KUKA KRL program: MyProgram_310().src

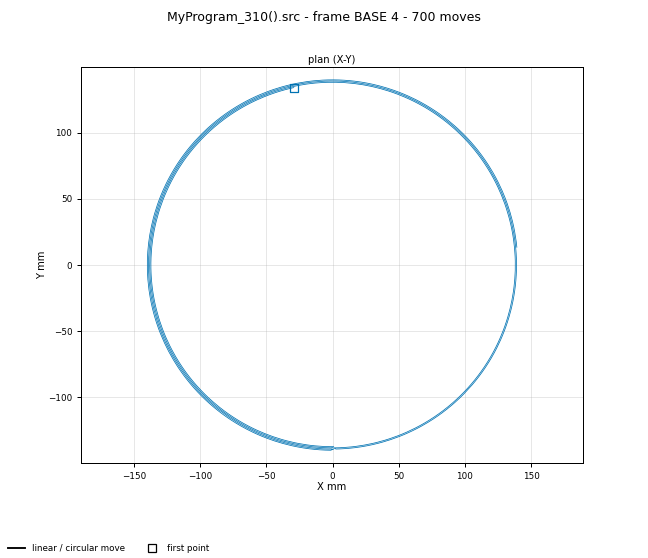
[picture p0: tool path of MyProgram_310().src in frame BASE 4, 700 of 700 moves have a stored position in this frame; points joined in program order, loops and branches not executed]
&ACCESS RVP
&REL 1
&PARAM TEMPLATE = C:\KRC\Roboter\Template\vorgabe
&PARAM EDITMASK = *
DEF MyProgram_310()
; ---- Setting reference (Base) ----
$BASE = BASE_DATA[4]

; --------------------------
; ---- Setting tool (TCP) ----
$TOOL = TOOL_DATA[3]
; --------------------------

$VEL.CP = VEL_APROX_PRINT
Startdeposition()
$VEL.CP = VEL_PRINT
LIN {X -29.2639,Y 134.0038,Z 182,A 103.6048,B 4.4109,C 0.0734,E1 4.3789,E2 349.3713} C_DIS
LIN {X -32.3216,Y 133.299,Z 182,A 104.9504,B 4.4109,C 0.0739,E1 4.3753,E2 348.0222} C_DIS
LIN {X -35.8759,Y 132.3877,Z 182,A 106.6346,B 4.4109,C 0.0736,E1 4.3707,E2 346.3204} C_DIS
LIN {X -40.2763,Y 131.1148,Z 182,A 108.4348,B 4.4108,C 0.076,E1 4.3659,E2 344.5352} C_DIS
LIN {X -43.6422,Y 130.0335,Z 182,A 110.3943,B 4.4108,C 0.0731,E1 4.3605,E2 342.5172} C_DIS
LIN {X -47.686,Y 128.606,Z 182,A 111.5731,B 4.4108,C 0.0799,E1 4.3576,E2 341.4149} C_DIS
LIN {X -51.93,Y 126.9528,Z 182,A 113.9515,B 4.4108,C 0.0778,E1 4.3513,E2 338.9794} C_DIS
LIN {X -54.9246,Y 125.6853,Z 182,A 115.0053,B 4.4107,C 0.0818,E1 4.3487,E2 337.964} C_DIS
LIN {X -57.8291,Y 124.3748,Z 182,A 116.3918,B 4.4107,C 0.0828,E1 4.3452,E2 336.5716} C_DIS
LIN {X -61.4347,Y 122.6365,Z 182,A 118.0932,B 4.4107,C 0.0846,E1 4.3409,E2 334.8678} C_DIS
LIN {X -64.5583,Y 121.0213,Z 182,A 119.5331,B 4.4106,C 0.0867,E1 4.3374,E2 333.4325} C_DIS
LIN {X -67.7824,Y 119.245,Z 182,A 121.2234,B 4.4106,C 0.0875,E1 4.3332,E2 331.7246} C_DIS
LIN {X -71.6244,Y 116.9775,Z 182,A 123.3545,B 4.4106,C 0.0881,E1 4.328,E2 329.5618} C_DIS
LIN {X -74.5849,Y 115.1125,Z 182,A 124.6005,B 4.4105,C 0.0919,E1 4.3252,E2 328.3436} C_DIS
LIN {X -78.3354,Y 112.5937,Z 182,A 126.5047,B 4.4105,C 0.0947,E1 4.3208,E2 326.4387} C_DIS
LIN {X -81.9968,Y 109.956,Z 182,A 128.4347,B 4.4104,C 0.0975,E1 4.3164,E2 324.5045} C_DIS
LIN {X -85.5745,Y 107.1952,Z 182,A 130.371,B 4.4103,C 0.1003,E1 4.3121,E2 322.5637} C_DIS
LIN {X -89.1427,Y 104.2473,Z 182,A 132.3771,B 4.4103,C 0.1033,E1 4.3078,E2 320.5502} C_DIS
LIN {X -92.5611,Y 101.2242,Z 182,A 134.3112,B 4.4101,C 0.1066,E1 4.3038,E2 318.6141} C_DIS
LIN {X -95.8331,Y 98.1319,Z 182,A 136.1996,B 4.4101,C 0.1102,E1 4.3,E2 316.7263} C_DIS
LIN {X -98.9014,Y 95.0391,Z 182,A 138.1181,B 4.41,C 0.1131,E1 4.2963,E2 314.7971} C_DIS
LIN {X -101.9762,Y 91.7318,Z 182,A 140.0414,B 4.4099,C 0.1167,E1 4.2926,E2 312.8707} C_DIS
LIN {X -104.9444,Y 88.3204,Z 182,A 141.957,B 4.4098,C 0.1206,E1 4.2891,E2 310.9533} C_DIS
LIN {X -107.7995,Y 84.8119,Z 182,A 143.9009,B 4.4097,C 0.1243,E1 4.2857,E2 309.0042} C_DIS
LIN {X -110.6043,Y 81.1202,Z 182,A 145.847,B 4.4096,C 0.1286,E1 4.2825,E2 307.0586} C_DIS
LIN {X -112.9805,Y 77.7767,Z 182,A 147.6562,B 4.4095,C 0.1319,E1 4.2796,E2 305.2389} C_DIS
LIN {X -115.8244,Y 73.475,Z 182,A 149.8731,B 4.4093,C 0.1366,E1 4.2762,E2 303.016} C_DIS
LIN {X -117.6466,Y 70.5207,Z 182,A 151.3055,B 4.4093,C 0.1402,E1 4.2741,E2 301.587} C_DIS
LIN {X -119.7774,Y 66.8381,Z 182,A 153.2138,B 4.4091,C 0.1437,E1 4.2715,E2 299.6639} C_DIS
LIN {X -121.98,Y 62.7249,Z 182,A 155.3274,B 4.409,C 0.1474,E1 4.2687,E2 297.5313} C_DIS
LIN {X -123.966,Y 58.7016,Z 182,A 157.0165,B 4.4088,C 0.1535,E1 4.2667,E2 295.8668} C_DIS
LIN {X -125.3677,Y 55.6446,Z 182,A 158.4571,B 4.4086,C 0.1568,E1 4.2651,E2 294.423} C_DIS
LIN {X -126.6541,Y 52.65,Z 182,A 159.7976,B 4.4086,C 0.1605,E1 4.2636,E2 293.0862} C_DIS
LIN {X -127.9591,Y 49.3944,Z 182,A 161.4133,B 4.4084,C 0.1634,E1 4.2619,E2 291.4528} C_DIS
LIN {X -130.0899,Y 43.4728,Z 182,A 164.1548,B 4.4082,C 0.1697,E1 4.2594,E2 288.6995} C_DIS
LIN {X -131.194,Y 40.0177,Z 182,A 166.0837,B 4.4082,C 0.171,E1 4.2578,E2 286.7197} C_DIS
LIN {X -132.3301,Y 36.0919,Z 182,A 167.3879,B 4.4078,C 0.1784,E1 4.2568,E2 285.4677} C_DIS
LIN {X -133.024,Y 33.4363,Z 182,A 168.6291,B 4.4078,C 0.1809,E1 4.256,E2 284.2155} C_DIS
LIN {X -133.8628,Y 29.9076,Z 182,A 170.2807,B 4.4076,C 0.1842,E1 4.2549,E2 282.548} C_DIS
LIN {X -134.7576,Y 25.568,Z 182,A 172.1099,B 4.4074,C 0.1895,E1 4.2539,E2 280.7228} C_DIS
LIN {X -135.4848,Y 21.3857,Z 182,A 173.9614,B 4.4072,C 0.1939,E1 4.2531,E2 278.863} C_DIS
LIN {X -135.9927,Y 17.8699,Z 182,A 175.4529,B 4.407,C 0.198,E1 4.2525,E2 277.3716} C_DIS
LIN {X -136.4492,Y 13.9804,Z 182,A 177.2549,B 4.4068,C 0.2016,E1 4.252,E2 275.5499} C_DIS
LIN {X -136.8021,Y 9.9275,Z 182,A 178.9425,B 4.4066,C 0.2064,E1 4.2516,E2 273.865} C_DIS
LIN {X -137.0448,Y 5.6759,Z 182,A -179.2169,B 4.4064,C 0.2111,E1 4.2513,E2 272.0179} C_DIS
LIN {X -137.1521,Y 1.7268,Z 182,A -177.4633,B 4.4062,C 0.2151,E1 4.2513,E2 270.2524} C_DIS
LIN {X -137.1387,Y -2.5339,Z 182,A -175.7226,B 4.4059,C 0.2204,E1 4.2513,E2 268.5179} C_DIS
LIN {X -137.0026,Y -6.6138,Z 182,A -173.9481,B 4.4057,C 0.2247,E1 4.2515,E2 266.7359} C_DIS
LIN {X -136.7867,Y -10.1386,Z 182,A -172.3669,B 4.4055,C 0.2282,E1 4.2518,E2 265.1422} C_DIS
LIN {X -136.3688,Y -14.7275,Z 182,A -170.4483,B 4.4052,C 0.2337,E1 4.2523,E2 263.2256} C_DIS
LIN {X -135.9713,Y -18.0329,Z 182,A -169.0247,B 4.4051,C 0.2373,E1 4.2528,E2 261.7988} C_DIS
LIN {X -135.4736,Y -21.4582,Z 182,A -167.5007,B 4.4049,C 0.2409,E1 4.2535,E2 260.2658} C_DIS
LIN {X -134.7446,Y -25.6362,Z 182,A -165.6181,B 4.4046,C 0.245,E1 4.2544,E2 258.3701} C_DIS
LIN {X -133.9141,Y -29.6793,Z 182,A -163.7588,B 4.4044,C 0.2489,E1 4.2555,E2 256.4946} C_DIS
LIN {X -132.9848,Y -33.5908,Z 182,A -162.1525,B 4.4041,C 0.254,E1 4.2566,E2 254.8986} C_DIS
LIN {X -131.3512,Y -39.504,Z 182,A -159.5891,B 4.4037,C 0.2609,E1 4.2585,E2 252.3367} C_DIS
LIN {X -130.4365,Y -42.4276,Z 182,A -158.0502,B 4.4037,C 0.2626,E1 4.2599,E2 250.7652} C_DIS
LIN {X -128.3433,Y -48.3872,Z 182,A -155.435,B 4.4032,C 0.2697,E1 4.2623,E2 248.1543} C_DIS
LIN {X -127.0767,Y -51.6226,Z 182,A -153.9839,B 4.403,C 0.2735,E1 4.2638,E2 246.704} C_DIS
LIN {X -125.713,Y -54.8607,Z 182,A -152.4663,B 4.4027,C 0.2769,E1 4.2655,E2 245.1807} C_DIS
LIN {X -124.3115,Y -57.9661,Z 182,A -150.9211,B 4.4026,C 0.2797,E1 4.2673,E2 243.6205} C_DIS
LIN {X -122.8733,Y -60.9546,Z 182,A -149.5531,B 4.4023,C 0.2832,E1 4.269,E2 242.2553} C_DIS
LIN {X -120.9706,Y -64.6528,Z 182,A -147.665,B 4.4021,C 0.2865,E1 4.2715,E2 240.3485} C_DIS
LIN {X -118.3587,Y -69.3183,Z 182,A -145.4078,B 4.4018,C 0.2917,E1 4.2746,E2 238.0892} C_DIS
LIN {X -116.1413,Y -72.9729,Z 182,A -143.5209,B 4.4016,C 0.2952,E1 4.2774,E2 236.1898} C_DIS
LIN {X -113.5739,Y -76.9074,Z 182,A -141.5681,B 4.4013,C 0.2998,E1 4.2804,E2 234.239} C_DIS
LIN {X -111.1027,Y -80.4362,Z 182,A -139.7071,B 4.401,C 0.3034,E1 4.2834,E2 232.3706} C_DIS
LIN {X -108.5628,Y -83.8329,Z 182,A -137.8763,B 4.4008,C 0.3068,E1 4.2866,E2 230.5326} C_DIS
LIN {X -105.8429,Y -87.2419,Z 182,A -135.969,B 4.4005,C 0.3101,E1 4.2899,E2 228.6148} C_DIS
LIN {X -102.8901,Y -90.7052,Z 182,A -133.4318,B 4.4006,C 0.3091,E1 4.2948,E2 225.9948} C_DIS
LIN {X -99.1771,Y -94.7506,Z 182,A -131.9418,B 4.3998,C 0.3199,E1 4.2974,E2 224.6103} C_DIS
LIN {X -96.5033,Y -97.4727,Z 182,A -130.2609,B 4.3997,C 0.3223,E1 4.3007,E2 222.9185} C_DIS
LIN {X -93.9205,Y -99.9639,Z 182,A -128.5538,B 4.3996,C 0.3235,E1 4.3042,E2 221.1845} C_DIS
LIN {X -90.6366,Y -102.9507,Z 182,A -126.441,B 4.3995,C 0.3247,E1 4.3087,E2 219.0381} C_DIS
LIN {X -88.135,Y -105.0999,Z 182,A -125.3023,B 4.3992,C 0.3291,E1 4.3111,E2 217.9309} C_DIS
LIN {X -85.5334,Y -107.2279,Z 182,A -123.8007,B 4.399,C 0.3306,E1 4.3144,E2 216.4166} C_DIS
LIN {X -81.9056,Y -110.0238,Z 182,A -121.8898,B 4.3988,C 0.3337,E1 4.3186,E2 214.5062} C_DIS
LIN {X -78.4854,Y -112.4894,Z 182,A -120.0573,B 4.3987,C 0.3359,E1 4.3228,E2 212.6644} C_DIS
LIN {X -74.8068,Y -114.9684,Z 182,A -118.1768,B 4.3985,C 0.3383,E1 4.3272,E2 210.7803} C_DIS
LIN {X -71.0909,Y -117.3025,Z 182,A -116.3724,B 4.3982,C 0.3411,E1 4.3315,E2 208.9797} C_DIS
LIN {X -67.5199,Y -119.3942,Z 182,A -114.5341,B 4.3982,C 0.3424,E1 4.336,E2 207.1269} C_DIS
LIN {X -63.7403,Y -121.4512,Z 182,A -112.8171,B 4.3979,C 0.3453,E1 4.3402,E2 205.4203} C_DIS
LIN {X -60.4027,Y -123.1455,Z 182,A -111.239,B 4.3978,C 0.347,E1 4.3442,E2 203.8401} C_DIS
LIN {X -57.3207,Y -124.6099,Z 182,A -109.8007,B 4.3977,C 0.3484,E1 4.3478,E2 202.3999} C_DIS
LIN {X -53.687,Y -126.2204,Z 182,A -108.1254,B 4.3976,C 0.35,E1 4.3521,E2 200.7225} C_DIS
LIN {X -51.231,Y -127.2345,Z 182,A -106.9551,B 4.3976,C 0.3505,E1 4.3551,E2 199.544} C_DIS
LIN {X -47.5863,Y -128.6433,Z 182,A -105.3745,B 4.3974,C 0.3524,E1 4.3593,E2 197.9699} C_DIS
LIN {X -44.8972,Y -129.6052,Z 182,A -104.1531,B 4.3974,C 0.3531,E1 4.3625,E2 196.7446} C_DIS
LIN {X -40.9503,Y -130.9084,Z 182,A -102.4109,B 4.3972,C 0.3543,E1 4.3671,E2 195.0012} C_DIS
LIN {X -38.449,Y -131.6623,Z 182,A -101.2729,B 4.3972,C 0.3546,E1 4.3702,E2 193.8567} C_DIS
LIN {X -34.9989,Y -132.6216,Z 182,A -99.7719,B 4.3972,C 0.3555,E1 4.3742,E2 192.3547} C_DIS
LIN {X -31.6937,Y -133.4504,Z 182,A -98.3727,B 4.397,C 0.3565,E1 4.378,E2 190.9583} C_DIS
LIN {X -28.7459,Y -134.1157,Z 182,A -97.1167,B 4.397,C 0.3571,E1 4.3815,E2 189.7027} C_DIS
LIN {X -25.5139,Y -134.768,Z 182,A -95.7025,B 4.397,C 0.3573,E1 4.3854,E2 188.2832} C_DIS
LIN {X -19.2093,Y -135.81,Z 182,A -93.1879,B 4.3968,C 0.3597,E1 4.3923,E2 185.7881} C_DIS
LIN {X -16.3537,Y -136.1834,Z 182,A -91.8444,B 4.3968,C 0.3586,E1 4.396,E2 184.4258} C_DIS
LIN {X -12.7776,Y -136.5657,Z 182,A -89.9841,B 4.3971,C 0.3552,E1 4.4013,E2 182.5175} C_DIS
LIN {X -9.1426,Y -136.8586,Z 182,A -88.7743,B 4.3969,C 0.3585,E1 4.4046,E2 181.3486} C_DIS
LIN {X -6.5538,Y -137.0056,Z 182,A -87.615,B 4.3969,C 0.3577,E1 4.4079,E2 180.1787} C_DIS
LIN {X -2.1717,Y -137.1447,Z 182,A -85.8504,B 4.3969,C 0.3582,E1 4.4128,E2 178.4221} C_DIS
LIN {X 0.9727,Y -137.1551,Z 182,A -84.8175,B 4.3967,C 0.3609,E1 4.4156,E2 177.4255} C_DIS
Enddeposition()
LIN {X 0.9727,Y -137.1551,Z 182,A -84.8175,B 4.3967,C 0.3609,E1 4.4156,E2 177.4255} C_DIS
Startdeposition()
$VEL.CP = VEL_PRINT
LIN {X -0.8195,Y -138.061,Z 182,A -85.9153,B 4.3834,C 0.3668,E1 4.3995,E2 178.6059} C_DIS
LIN {X -4.6066,Y -137.9886,Z 182,A -87.4496,B 4.3834,C 0.3665,E1 4.3952,E2 180.136} C_DIS
LIN {X -7.7094,Y -137.8501,Z 182,A -88.741,B 4.3834,C 0.3665,E1 4.3916,E2 181.4282} C_DIS
LIN {X -10.3826,Y -137.6727,Z 182,A -89.8567,B 4.3834,C 0.3665,E1 4.3885,E2 182.5448} C_DIS
LIN {X -13.4072,Y -137.4109,Z 182,A -91.1307,B 4.3834,C 0.3665,E1 4.3849,E2 183.8213} C_DIS
LIN {X -16.6884,Y -137.0513,Z 182,A -92.5339,B 4.3834,C 0.3665,E1 4.381,E2 185.2293} C_DIS
LIN {X -20.3271,Y -136.5609,Z 182,A -94.0261,B 4.3834,C 0.3658,E1 4.3769,E2 186.718} C_DIS
LIN {X -23.5214,Y -136.0471,Z 182,A -95.3761,B 4.3834,C 0.3654,E1 4.3732,E2 188.0694} C_DIS
LIN {X -26.161,Y -135.5621,Z 182,A -96.5101,B 4.3834,C 0.3652,E1 4.37,E2 189.2064} C_DIS
LIN {X -29.4753,Y -134.8804,Z 182,A -97.9114,B 4.3835,C 0.3645,E1 4.3662,E2 190.6077} C_DIS
LIN {X -33.1585,Y -134.0246,Z 182,A -99.4918,B 4.3836,C 0.3638,E1 4.3619,E2 192.1901} C_DIS
LIN {X -35.7982,Y -133.3414,Z 182,A -100.6484,B 4.3836,C 0.3634,E1 4.3588,E2 193.3503} C_DIS
LIN {X -39.0801,Y -132.4168,Z 182,A -102.0677,B 4.3837,C 0.3625,E1 4.355,E2 194.7704} C_DIS
LIN {X -42.3518,Y -131.4071,Z 182,A -103.5367,B 4.3837,C 0.3619,E1 4.351,E2 196.2461} C_DIS
LIN {X -46.0263,Y -130.1678,Z 182,A -105.1218,B 4.3839,C 0.3604,E1 4.3468,E2 197.8284} C_DIS
LIN {X -48.8301,Y -129.1401,Z 182,A -106.3786,B 4.3839,C 0.3595,E1 4.3435,E2 199.0878} C_DIS
LIN {X -52.4126,Y -127.7302,Z 182,A -107.9924,B 4.3841,C 0.3581,E1 4.3394,E2 200.7039} C_DIS
LIN {X -55.1251,Y -126.5808,Z 182,A -109.2309,B 4.3841,C 0.3571,E1 4.3362,E2 201.9447} C_DIS
LIN {X -58.2734,Y -125.1626,Z 182,A -110.6836,B 4.3843,C 0.3557,E1 4.3325,E2 203.4002} C_DIS
LIN {X -61.8592,Y -123.4323,Z 182,A -112.5047,B 4.3843,C 0.3553,E1 4.3279,E2 205.2436} C_DIS
LIN {X -65.7297,Y -121.4154,Z 182,A -114.2523,B 4.3845,C 0.3526,E1 4.3236,E2 206.983} C_DIS
LIN {X -69.3881,Y -119.3618,Z 182,A -116.0516,B 4.3847,C 0.3508,E1 4.3192,E2 208.7899} C_DIS
LIN {X -73.1029,Y -117.1234,Z 182,A -117.7965,B 4.3849,C 0.3479,E1 4.315,E2 210.5277} C_DIS
LIN {X -76.2241,Y -115.1169,Z 182,A -119.4346,B 4.385,C 0.3465,E1 4.3112,E2 212.1786} C_DIS
LIN {X -79.7324,Y -112.7149,Z 182,A -121.1604,B 4.3852,C 0.3435,E1 4.3072,E2 213.8993} C_DIS
LIN {X -82.8118,Y -110.473,Z 182,A -122.8802,B 4.3854,C 0.3421,E1 4.3033,E2 215.6372} C_DIS
LIN {X -86.3289,Y -107.747,Z 182,A -124.7605,B 4.3856,C 0.3393,E1 4.2992,E2 217.5217} C_DIS
LIN {X -89.7623,Y -104.9038,Z 182,A -126.598,B 4.3858,C 0.336,E1 4.2953,E2 219.3573} C_DIS
LIN {X -92.9151,Y -102.121,Z 182,A -128.3263,B 4.3861,C 0.3327,E1 4.2917,E2 221.0832} C_DIS
LIN {X -95.7133,Y -99.504,Z 182,A -130.0151,B 4.3862,C 0.3305,E1 4.2882,E2 222.7846} C_DIS
LIN {X -98.785,Y -96.4547,Z 182,A -131.8688,B 4.3865,C 0.3275,E1 4.2846,E2 224.6454} C_DIS
LIN {X -101.7729,Y -93.2963,Z 182,A -133.6694,B 4.3867,C 0.3239,E1 4.2811,E2 226.4451} C_DIS
LIN {X -104.3215,Y -90.4384,Z 182,A -135.3449,B 4.3869,C 0.3212,E1 4.278,E2 228.1314} C_DIS
LIN {X -107.1876,Y -87.0224,Z 182,A -137.2238,B 4.3872,C 0.3175,E1 4.2747,E2 230.0136} C_DIS
LIN {X -109.7812,Y -83.7258,Z 182,A -138.9788,B 4.3875,C 0.3138,E1 4.2717,E2 231.7698} C_DIS
LIN {X -112.2673,Y -80.3613,Z 182,A -140.8085,B 4.3877,C 0.3107,E1 4.2686,E2 233.6111} C_DIS
LIN {X -114.7245,Y -76.8128,Z 182,A -142.6406,B 4.388,C 0.3069,E1 4.2658,E2 235.4478} C_DIS
LIN {X -117.0649,Y -73.1968,Z 182,A -144.4981,B 4.3882,C 0.3032,E1 4.263,E2 237.3137} C_DIS
LIN {X -119.267,Y -69.5519,Z 182,A -146.2815,B 4.3885,C 0.2991,E1 4.2604,E2 239.0986} C_DIS
LIN {X -121.4154,Y -65.7297,Z 182,A -148.2159,B 4.3887,C 0.2955,E1 4.2578,E2 241.047} C_DIS
LIN {X -123.2037,Y -62.3081,Z 182,A -149.74,B 4.389,C 0.2909,E1 4.2558,E2 242.5603} C_DIS
LIN {X -124.9503,Y -58.7325,Z 182,A -151.4376,B 4.3893,C 0.2871,E1 4.2538,E2 244.2632} C_DIS
LIN {X -126.2793,Y -55.8143,Z 182,A -152.7859,B 4.3895,C 0.2838,E1 4.2522,E2 245.613} C_DIS
LIN {X -127.5386,Y -52.8713,Z 182,A -154.1755,B 4.3897,C 0.2808,E1 4.2507,E2 247.0099} C_DIS
LIN {X -128.8126,Y -49.687,Z 182,A -155.6413,B 4.3899,C 0.2774,E1 4.2492,E2 248.4803} C_DIS
LIN {X -130.001,Y -46.489,Z 182,A -157.1006,B 4.3901,C 0.274,E1 4.2478,E2 249.9445} C_DIS
LIN {X -131.0722,Y -43.3763,Z 182,A -158.5205,B 4.3903,C 0.2707,E1 4.2465,E2 251.3705} C_DIS
LIN {X -132.2647,Y -39.5998,Z 182,A -160.2028,B 4.3906,C 0.2665,E1 4.2452,E2 253.057} C_DIS
LIN {X -133.1864,Y -36.3794,Z 182,A -161.6362,B 4.3908,C 0.2631,E1 4.2441,E2 254.495} C_DIS
LIN {X -133.8647,Y -33.7887,Z 182,A -162.7816,B 4.391,C 0.2603,E1 4.2433,E2 255.6441} C_DIS
LIN {X -134.6625,Y -30.4548,Z 182,A -164.2614,B 4.3912,C 0.2567,E1 4.2423,E2 257.1304} C_DIS
LIN {X -135.4539,Y -26.7266,Z 182,A -165.8816,B 4.3914,C 0.2526,E1 4.2414,E2 258.7546} C_DIS
LIN {X -135.9643,Y -23.9842,Z 182,A -167.0752,B 4.3916,C 0.2497,E1 4.2408,E2 259.952} C_DIS
LIN {X -136.4895,Y -20.7882,Z 182,A -168.4619,B 4.3918,C 0.2462,E1 4.2402,E2 261.3432} C_DIS
LIN {X -136.9365,Y -17.6054,Z 182,A -169.8781,B 4.3919,C 0.243,E1 4.2397,E2 262.769} C_DIS
LIN {X -137.3066,Y -14.4381,Z 182,A -171.204,B 4.3921,C 0.2393,E1 4.2393,E2 264.0944} C_DIS
LIN {X -137.5888,Y -11.4373,Z 182,A -172.5095,B 4.3923,C 0.2361,E1 4.239,E2 265.4059} C_DIS
LIN {X -137.8075,Y -8.4003,Z 182,A -173.8339,B 4.3925,C 0.233,E1 4.2387,E2 266.7372} C_DIS
LIN {X -137.9712,Y -5.0541,Z 182,A -175.2723,B 4.3927,C 0.2293,E1 4.2385,E2 268.1807} C_DIS
LIN {X -138.0618,Y -0.8135,Z 182,A -177.0703,B 4.3929,C 0.2246,E1 4.2385,E2 269.9822} C_DIS
LIN {X -138.0434,Y 2.3508,Z 182,A -178.4274,B 4.3931,C 0.2212,E1 4.2385,E2 271.3439} C_DIS
LIN {X -137.9448,Y 5.7297,Z 182,A -179.9008,B 4.3933,C 0.2177,E1 4.2386,E2 272.8252} C_DIS
LIN {X -137.754,Y 9.2695,Z 182,A 178.6109,B 4.3935,C 0.2136,E1 4.2389,E2 274.3147} C_DIS
LIN {X -137.5453,Y 11.9519,Z 182,A 177.4146,B 4.3935,C 0.211,E1 4.2392,E2 275.5201} C_DIS
LIN {X -137.0709,Y 16.5243,Z 182,A 175.4536,B 4.3938,C 0.2059,E1 4.2398,E2 277.4863} C_DIS
LIN {X -136.6041,Y 20.0248,Z 182,A 173.9413,B 4.394,C 0.2021,E1 4.2404,E2 279.0034} C_DIS
LIN {X -136.0471,Y 23.5214,Z 182,A 172.439,B 4.3942,C 0.1982,E1 4.241,E2 280.5088} C_DIS
LIN {X -135.4539,Y 26.7266,Z 182,A 171.0385,B 4.3943,C 0.1948,E1 4.2418,E2 281.9142} C_DIS
LIN {X -134.905,Y 29.3618,Z 182,A 169.8668,B 4.3945,C 0.192,E1 4.2425,E2 283.0918} C_DIS
LIN {X -134.0246,Y 33.1585,Z 182,A 168.209,B 4.3946,C 0.1878,E1 4.2435,E2 284.7535} C_DIS
LIN {X -133.3105,Y 35.914,Z 182,A 166.9863,B 4.3948,C 0.1849,E1 4.2444,E2 285.9803} C_DIS
LIN {X -132.4154,Y 39.0851,Z 182,A 165.5801,B 4.3949,C 0.1814,E1 4.2455,E2 287.3902} C_DIS
LIN {X -131.4071,Y 42.3518,Z 182,A 164.0634,B 4.395,C 0.1782,E1 4.2468,E2 288.918} C_DIS
LIN {X -130.1678,Y 46.0263,Z 182,A 162.4427,B 4.3952,C 0.174,E1 4.2483,E2 290.5389} C_DIS
LIN {X -128.9918,Y 49.2261,Z 182,A 160.9811,B 4.3953,C 0.1705,E1 4.2497,E2 292.0052} C_DIS
LIN {X -127.7302,Y 52.4126,Z 182,A 159.5121,B 4.3955,C 0.1671,E1 4.2512,E2 293.4789} C_DIS
LIN {X -126.602,Y 55.0761,Z 182,A 158.2661,B 4.3955,C 0.1643,E1 4.2526,E2 294.7295} C_DIS
LIN {X -125.1604,Y 58.2781,Z 182,A 156.7688,B 4.3957,C 0.1608,E1 4.2544,E2 296.2306} C_DIS
LIN {X -123.6547,Y 61.4083,Z 182,A 155.2388,B 4.3958,C 0.1577,E1 4.2563,E2 297.7703} C_DIS
LIN {X -121.7097,Y 65.1819,Z 182,A 153.3744,B 4.396,C 0.154,E1 4.2587,E2 299.6461} C_DIS
LIN {X -119.5507,Y 69.0619,Z 182,A 151.4737,B 4.396,C 0.1499,E1 4.2613,E2 301.5523} C_DIS
LIN {X -117.4547,Y 72.5706,Z 182,A 149.8211,B 4.3962,C 0.1455,E1 4.2637,E2 303.1982} C_DIS
LIN {X -115.2806,Y 75.9755,Z 182,A 148.0718,B 4.3964,C 0.142,E1 4.2664,E2 304.9551} C_DIS
LIN {X -112.9675,Y 79.3744,Z 182,A 146.2555,B 4.3964,C 0.1388,E1 4.2693,E2 306.7836} C_DIS
LIN {X -110.6264,Y 82.6058,Z 182,A 144.6421,B 4.3966,C 0.1348,E1 4.2719,E2 308.3903} C_DIS
LIN {X -108.3017,Y 85.632,Z 182,A 142.9232,B 4.3966,C 0.1322,E1 4.2749,E2 310.1247} C_DIS
LIN {X -105.4817,Y 89.0826,Z 182,A 141.0517,B 4.3968,C 0.1284,E1 4.2782,E2 311.9974} C_DIS
LIN {X -102.7198,Y 92.2526,Z 182,A 139.2931,B 4.3968,C 0.1248,E1 4.2815,E2 313.7562} C_DIS
LIN {X -99.7357,Y 95.4709,Z 182,A 137.3865,B 4.397,C 0.1217,E1 4.2852,E2 315.6718} C_DIS
LIN {X -96.5396,Y 98.7017,Z 182,A 135.5306,B 4.397,C 0.1178,E1 4.2888,E2 317.5225} C_DIS
LIN {X -93.7638,Y 101.3431,Z 182,A 133.9043,B 4.3971,C 0.115,E1 4.2921,E2 319.152} C_DIS
LIN {X -91.1109,Y 103.7347,Z 182,A 132.3179,B 4.3971,C 0.113,E1 4.2955,E2 320.75} C_DIS
LIN {X -87.8397,Y 106.5183,Z 182,A 130.4861,B 4.3973,C 0.1102,E1 4.2994,E2 322.5864} C_DIS
LIN {X -84.4316,Y 109.2393,Z 182,A 128.6902,B 4.3973,C 0.107,E1 4.3033,E2 324.3792} C_DIS
LIN {X -81.3829,Y 111.5299,Z 182,A 127.0473,B 4.3974,C 0.1049,E1 4.307,E2 326.0283} C_DIS
LIN {X -77.9699,Y 113.9413,Z 182,A 125.3115,B 4.3974,C 0.1021,E1 4.311,E2 327.7629} C_DIS
LIN {X -74.8095,Y 116.0414,Z 182,A 123.7393,B 4.3975,C 0.0997,E1 4.3147,E2 329.3337} C_DIS
LIN {X -71.2836,Y 118.2395,Z 182,A 121.9574,B 4.3975,C 0.0977,E1 4.319,E2 331.1213} C_DIS
LIN {X -67.8083,Y 120.2662,Z 182,A 120.1905,B 4.3975,C 0.0962,E1 4.3233,E2 332.899} C_DIS
LIN {X -63.8596,Y 122.4067,Z 182,A 118.4046,B 4.3977,C 0.0932,E1 4.3276,E2 334.6739} C_DIS
LIN {X -60.2989,Y 124.2019,Z 182,A 116.7273,B 4.3977,C 0.0914,E1 4.3318,E2 336.3529} C_DIS
LIN {X -57.4185,Y 125.5579,Z 182,A 115.375,B 4.3977,C 0.0901,E1 4.3353,E2 337.7081} C_DIS
LIN {X -54.382,Y 126.9021,Z 182,A 114.0038,B 4.3977,C 0.0886,E1 4.3388,E2 339.0775} C_DIS
LIN {X -51.2811,Y 128.1863,Z 182,A 112.5879,B 4.3977,C 0.0874,E1 4.3424,E2 340.4952} C_DIS
LIN {X -48.0895,Y 129.4175,Z 182,A 111.1542,B 4.3978,C 0.0861,E1 4.3462,E2 341.9297} C_DIS
LIN {X -44.8859,Y 130.5632,Z 182,A 109.7298,B 4.3978,C 0.085,E1 4.35,E2 343.3548} C_DIS
LIN {X -41.4038,Y 131.7099,Z 182,A 108.1872,B 4.3978,C 0.084,E1 4.3541,E2 344.899} C_DIS
LIN {X -37.9899,Y 132.736,Z 182,A 106.7053,B 4.3978,C 0.0829,E1 4.358,E2 346.3804} C_DIS
LIN {X -35.1003,Y 133.5275,Z 182,A 105.4796,B 4.3978,C 0.0819,E1 4.3613,E2 347.6031} C_DIS
LIN {X -32.0139,Y 134.3005,Z 182,A 104.0866,B 4.3978,C 0.0817,E1 4.3651,E2 349.0042} C_DIS
LIN {X -28.3324,Y 135.1272,Z 182,A 102.5528,B 4.3979,C 0.0806,E1 4.3693,E2 350.5333} C_DIS
LIN {X -25.5863,Y 135.6719,Z 182,A 101.3868,B 4.3979,C 0.0801,E1 4.3725,E2 351.699} C_DIS
LIN {X -22.3847,Y 136.2368,Z 182,A 100.0333,B 4.3979,C 0.0796,E1 4.3762,E2 353.0523} C_DIS
LIN {X -19.195,Y 136.7227,Z 182,A 98.6914,B 4.3979,C 0.0791,E1 4.3799,E2 354.3939} C_DIS
LIN {X -15.5617,Y 137.1857,Z 182,A 97.1686,B 4.3979,C 0.0787,E1 4.3842,E2 355.9164} C_DIS
LIN {X -12.8611,Y 137.4633,Z 182,A 96.022,B 4.3979,C 0.0787,E1 4.3874,E2 357.0647} C_DIS
LIN {X -9.2695,Y 137.754,Z 182,A 94.5461,B 4.3979,C 0.0783,E1 4.3915,E2 358.5376} C_DIS
LIN {X -6.6042,Y 137.9057,Z 182,A 93.4663,B 4.3979,C 0.0779,E1 4.3945,E2 359.6134} C_DIS
LIN {X -3.9025,Y 138.0082,Z 182,A 92.2784,B 4.3979,C 0.0785,E1 4.3978,E2 360.8088} C_DIS
LIN {X 0,Y 138.0655,Z 182,A 90.7024,B 4.3979,C 0.0782,E1 4.4022,E2 362.3789} C_DIS
LIN {X 2.6207,Y 138.0389,Z 182,A 89.5769,B 4.3979,C 0.0787,E1 4.4053,E2 363.5085} C_DIS
LIN {X 6.155,Y 137.9282,Z 182,A 88.1464,B 4.3979,C 0.0786,E1 4.4093,E2 364.9339} C_DIS
LIN {X 9.2695,Y 137.754,Z 182,A 86.8533,B 4.3979,C 0.0789,E1 4.4129,E2 366.2263} C_DIS
LIN {X 13.9815,Y 137.3557,Z 182,A 84.8946,B 4.3979,C 0.0795,E1 4.4184,E2 368.1839} C_DIS
LIN {X 16.6884,Y 137.0513,Z 182,A 83.7284,B 4.3979,C 0.0803,E1 4.4216,E2 369.3539} C_DIS
LIN {X 20.3271,Y 136.5609,Z 182,A 82.2489,B 4.3979,C 0.0805,E1 4.4257,E2 370.8276} C_DIS
LIN {X 22.9824,Y 136.1371,Z 182,A 81.0868,B 4.3979,C 0.0816,E1 4.4289,E2 371.995} C_DIS
LIN {X 26.7266,Y 135.4539,Z 182,A 79.5665,B 4.3979,C 0.0819,E1 4.4331,E2 373.5076} C_DIS
LIN {X 29.4753,Y 134.8804,Z 182,A 78.4076,B 4.3979,C 0.0826,E1 4.4362,E2 374.6653} C_DIS
LIN {X 33.0405,Y 134.053,Z 182,A 76.9042,B 4.3979,C 0.0836,E1 4.4403,E2 376.1665} C_DIS
LIN {X 35.914,Y 133.3105,Z 182,A 75.677,B 4.3979,C 0.0845,E1 4.4436,E2 377.3929} C_DIS
LIN {X 39.1345,Y 132.4009,Z 182,A 74.2999,B 4.3979,C 0.0855,E1 4.4473,E2 378.7681} C_DIS
LIN {X 42.3518,Y 131.4071,Z 182,A 72.8751,B 4.3978,C 0.0871,E1 4.4511,E2 380.196} C_DIS
LIN {X 45.7133,Y 130.2763,Z 182,A 71.4551,B 4.3978,C 0.088,E1 4.4549,E2 381.6094} C_DIS
LIN {X 49.2261,Y 128.9918,Z 182,A 69.9231,B 4.3978,C 0.0894,E1 4.4589,E2 383.1387} C_DIS
LIN {X 52.4126,Y 127.7302,Z 182,A 68.5172,B 4.3978,C 0.0908,E1 4.4625,E2 384.5424} C_DIS
LIN {X 55.0623,Y 126.608,Z 182,A 67.3295,B 4.3977,C 0.0922,E1 4.4656,E2 385.7291} C_DIS
LIN {X 58.2781,Y 125.1604,Z 182,A 65.8932,B 4.3977,C 0.0937,E1 4.4692,E2 387.162} C_DIS
LIN {X 61.8592,Y 123.4323,Z 182,A 64.1239,B 4.3976,C 0.0971,E1 4.4737,E2 388.9458} C_DIS
LIN {X 65.7297,Y 121.4154,Z 182,A 62.3567,B 4.3976,C 0.0991,E1 4.478,E2 390.7074} C_DIS
LIN {X 69.5519,Y 119.267,Z 182,A 60.691,B 4.3976,C 0.1001,E1 4.482,E2 392.3542} C_DIS
LIN {X 72.5706,Y 117.4547,Z 182,A 59.2411,B 4.3975,C 0.1022,E1 4.4855,E2 393.8028} C_DIS
LIN {X 76.076,Y 115.2144,Z 182,A 57.5258,B 4.3975,C 0.1048,E1 4.4895,E2 395.5167} C_DIS
LIN {X 79.217,Y 113.0785,Z 182,A 55.939,B 4.3973,C 0.1075,E1 4.4931,E2 397.1048} C_DIS
LIN {X 82.8118,Y 110.473,Z 182,A 54.1417,B 4.3973,C 0.1102,E1 4.4972,E2 398.8967} C_DIS
LIN {X 86.2542,Y 107.8064,Z 182,A 52.3605,B 4.3972,C 0.1131,E1 4.5011,E2 400.6748} C_DIS
LIN {X 89.6532,Y 104.9966,Z 182,A 50.5624,B 4.3972,C 0.1161,E1 4.5049,E2 402.4692} C_DIS
LIN {X 92.9151,Y 102.121,Z 182,A 48.8415,B 4.3971,C 0.1186,E1 4.5085,E2 404.18} C_DIS
LIN {X 95.8988,Y 99.3244,Z 182,A 47.1188,B 4.397,C 0.1223,E1 4.512,E2 405.9061} C_DIS
LIN {X 99.1246,Y 96.1051,Z 182,A 45.2833,B 4.3969,C 0.1255,E1 4.5155,E2 407.735} C_DIS
LIN {X 101.9476,Y 93.1062,Z 182,A 43.5891,B 4.3968,C 0.1289,E1 4.5188,E2 409.4277} C_DIS
LIN {X 104.9038,Y 89.7623,Z 182,A 41.8136,B 4.3967,C 0.132,E1 4.522,E2 411.1942} C_DIS
LIN {X 107.5853,Y 86.5293,Z 182,A 40.1606,B 4.3966,C 0.1348,E1 4.5249,E2 412.8364} C_DIS
LIN {X 109.9374,Y 83.5216,Z 182,A 38.5603,B 4.3965,C 0.1386,E1 4.5276,E2 414.4392} C_DIS
LIN {X 112.5672,Y 79.9419,Z 182,A 36.854,B 4.3964,C 0.1412,E1 4.5304,E2 416.1289} C_DIS
LIN {X 114.7245,Y 76.8128,Z 182,A 35.2409,B 4.3963,C 0.1453,E1 4.5329,E2 417.747} C_DIS
LIN {X 117.1234,Y 73.1029,Z 182,A 33.4702,B 4.3961,C 0.149,E1 4.5356,E2 419.5105} C_DIS
LIN {X 119.267,Y 69.5519,Z 182,A 31.8045,B 4.3961,C 0.1525,E1 4.5379,E2 421.17} C_DIS
LIN {X 121.4154,Y 65.7297,Z 182,A 29.9777,B 4.3958,C 0.1571,E1 4.5404,E2 422.9984} C_DIS
LIN {X 123.2037,Y 62.3081,Z 182,A 28.5009,B 4.3958,C 0.1596,E1 4.5423,E2 424.4601} C_DIS
LIN {X 124.9503,Y 58.7325,Z 182,A 26.9385,B 4.3956,C 0.1627,E1 4.5442,E2 426.0121} C_DIS
LIN {X 126.383,Y 55.5825,Z 182,A 25.5455,B 4.3956,C 0.1659,E1 4.5457,E2 427.4004} C_DIS
LIN {X 127.5386,Y 52.8713,Z 182,A 24.3598,B 4.3954,C 0.1686,E1 4.547,E2 428.5819} C_DIS
LIN {X 128.8126,Y 49.687,Z 182,A 22.9805,B 4.3953,C 0.1718,E1 4.5484,E2 429.9563} C_DIS
LIN {X 129.9939,Y 46.5087,Z 182,A 21.6144,B 4.3952,C 0.1751,E1 4.5497,E2 431.318} C_DIS
LIN {X 131.1041,Y 43.2805,Z 182,A 20.2053,B 4.395,C 0.1788,E1 4.551,E2 432.7269} C_DIS
LIN {X 132.2489,Y 39.6512,Z 182,A 18.7189,B 4.3949,C 0.1819,E1 4.5522,E2 434.2025} C_DIS
LIN {X 133.0573,Y 36.8411,Z 182,A 17.5024,B 4.3948,C 0.1852,E1 4.5531,E2 435.42} C_DIS
LIN {X 133.9065,Y 33.6238,Z 182,A 16.2037,B 4.3946,C 0.188,E1 4.554,E2 436.709} C_DIS
LIN {X 134.7801,Y 29.9399,Z 182,A 14.683,B 4.3945,C 0.1917,E1 4.555,E2 438.2244} C_DIS
LIN {X 135.4539,Y 26.7266,Z 182,A 13.3647,B 4.3943,C 0.1949,E1 4.5557,E2 439.5379} C_DIS
LIN {X 136.2368,Y 22.3847,Z 182,A 11.5943,B 4.3941,C 0.1992,E1 4.5565,E2 441.3016} C_DIS
LIN {X 136.7227,Y 19.195,Z 182,A 10.2997,B 4.394,C 0.2024,E1 4.5571,E2 442.5915} C_DIS
LIN {X 137.1857,Y 15.5617,Z 182,A 8.8294,B 4.3938,C 0.2061,E1 4.5576,E2 444.0565} C_DIS
LIN {X 137.4633,Y 12.8611,Z 182,A 7.7525,B 4.3938,C 0.2086,E1 4.5579,E2 445.1278} C_DIS
LIN {X 137.754,Y 9.2695,Z 182,A 6.2948,B 4.3935,C 0.2123,E1 4.5582,E2 446.5818} C_DIS
LIN {X 137.9057,Y 6.6042,Z 182,A 5.2247,B 4.3935,C 0.215,E1 4.5583,E2 447.6478} C_DIS
LIN {X 138.0315,Y 3.0645,Z 182,A 3.6488,B 4.3931,C 0.2205,E1 4.5584,E2 449.2382} C_DIS
LIN {X 138.0618,Y -0.8135,Z 182,A 2.1458,B 4.393,C 0.2237,E1 4.5584,E2 450.7287} C_DIS
LIN {X 138.004,Y -4.0532,Z 182,A 0.8886,B 4.3928,C 0.2264,E1 4.5584,E2 451.9758} C_DIS
LIN {X 137.8501,Y -7.7094,Z 182,A -0.5322,B 4.3927,C 0.2294,E1 4.5582,E2 453.3852} C_DIS
LIN {X 137.6727,Y -10.3826,Z 182,A -1.6118,B 4.3925,C 0.2322,E1 4.558,E2 454.4615} C_DIS
LIN {X 137.3557,Y -13.9815,Z 182,A -3.0654,B 4.3923,C 0.2358,E1 4.5576,E2 455.9104} C_DIS
LIN {X 137.0652,Y -16.5719,Z 182,A -4.1705,B 4.3922,C 0.2392,E1 4.5572,E2 457.0192} C_DIS
LIN {X 136.5609,Y -20.3271,Z 182,A -5.6407,B 4.392,C 0.2423,E1 4.5566,E2 458.4776} C_DIS
LIN {X 136.0471,Y -23.5214,Z 182,A -6.9434,B 4.3918,C 0.2455,E1 4.5561,E2 459.7762} C_DIS
LIN {X 135.4539,Y -26.7266,Z 182,A -8.2561,B 4.3916,C 0.2488,E1 4.5554,E2 461.0849} C_DIS
LIN {X 134.9226,Y -29.28,Z 182,A -9.3234,B 4.3915,C 0.2516,E1 4.5547,E2 462.151} C_DIS
LIN {X 134.0658,Y -32.9876,Z 182,A -10.845,B 4.3913,C 0.2553,E1 4.5538,E2 463.6665} C_DIS
LIN {X 133.3105,Y -35.914,Z 182,A -12.0567,B 4.3911,C 0.2582,E1 4.5529,E2 464.8737} C_DIS
LIN {X 132.4009,Y -39.1345,Z 182,A -13.4046,B 4.3909,C 0.2614,E1 4.5519,E2 466.2175} C_DIS
LIN {X 131.4071,Y -42.3518,Z 182,A -14.8004,B 4.3907,C 0.2652,E1 4.5507,E2 467.6142} C_DIS
LIN {X 130.1678,Y -46.0263,Z 182,A -16.3234,B 4.3905,C 0.2685,E1 4.5493,E2 469.1275} C_DIS
LIN {X 128.9918,Y -49.2261,Z 182,A -17.6975,B 4.3903,C 0.2717,E1 4.548,E2 470.4974} C_DIS
LIN {X 127.7302,Y -52.4126,Z 182,A -19.0792,B 4.3901,C 0.275,E1 4.5465,E2 471.8751} C_DIS
LIN {X 126.6172,Y -55.0409,Z 182,A -20.241,B 4.3899,C 0.2778,E1 4.5453,E2 473.0349} C_DIS
LIN {X 125.1604,Y -58.2781,Z 182,A -21.6618,B 4.3897,C 0.281,E1 4.5436,E2 474.4502} C_DIS
LIN {X 123.4323,Y -61.8592,Z 182,A -23.405,B 4.3893,C 0.2865,E1 4.5414,E2 476.2069} C_DIS
LIN {X 121.447,Y -65.6708,Z 182,A -25.0776,B 4.3891,C 0.2896,E1 4.5393,E2 477.8667} C_DIS
LIN {X 119.267,Y -69.5519,Z 182,A -26.8559,B 4.3889,C 0.2933,E1 4.5368,E2 479.6376} C_DIS
LIN {X 117.1234,Y -73.1029,Z 182,A -28.5253,B 4.3886,C 0.2969,E1 4.5344,E2 481.3017} C_DIS
LIN {X 114.683,Y -76.875,Z 182,A -30.3672,B 4.3883,C 0.3011,E1 4.5316,E2 483.1423} C_DIS
LIN {X 112.2002,Y -80.4552,Z 182,A -32.0473,B 4.3882,C 0.3038,E1 4.5289,E2 484.8072} C_DIS
LIN {X 110.0922,Y -83.3165,Z 182,A -33.5158,B 4.3879,C 0.3072,E1 4.5264,E2 486.2762} C_DIS
LIN {X 107.5513,Y -86.5714,Z 182,A -35.2442,B 4.3876,C 0.3113,E1 4.5234,E2 488.0079} C_DIS
LIN {X 104.9038,Y -89.7623,Z 182,A -36.8927,B 4.3874,C 0.3142,E1 4.5205,E2 489.6485} C_DIS
LIN {X 102.121,Y -92.9151,Z 182,A -38.5351,B 4.3873,C 0.3167,E1 4.5174,E2 491.279} C_DIS
LIN {X 99.504,Y -95.7133,Z 182,A -40.1475,B 4.387,C 0.3204,E1 4.5143,E2 492.8956} C_DIS
LIN {X 96.5396,Y -98.7017,Z 182,A -41.793,B 4.3868,C 0.3228,E1 4.5111,E2 494.5294} C_DIS
LIN {X 93.7638,Y -101.3431,Z 182,A -43.4074,B 4.3866,C 0.3263,E1 4.5078,E2 496.1483} C_DIS
LIN {X 90.6327,Y -104.1519,Z 182,A -45.0855,B 4.3864,C 0.3289,E1 4.5043,E2 497.8189} C_DIS
LIN {X 87.4736,Y -106.8189,Z 182,A -46.8229,B 4.3861,C 0.3324,E1 4.5006,E2 499.5606} C_DIS
LIN {X 83.9733,Y -109.5919,Z 182,A -48.6343,B 4.3859,C 0.3353,E1 4.4966,E2 501.368} C_DIS
LIN {X 80.4552,Y -112.2002,Z 182,A -50.4085,B 4.3857,C 0.338,E1 4.4926,E2 503.138} C_DIS
LIN {X 76.8128,Y -114.7245,Z 182,A -52.2141,B 4.3855,C 0.3407,E1 4.4884,E2 504.9407} C_DIS
LIN {X 73.1029,Y -117.1234,Z 182,A -53.995,B 4.3853,C 0.343,E1 4.4842,E2 506.7162} C_DIS
LIN {X 69.5519,Y -119.267,Z 182,A -55.6778,B 4.3851,C 0.3453,E1 4.4802,E2 508.3953} C_DIS
LIN {X 65.7297,Y -121.4154,Z 182,A -57.5255,B 4.3849,C 0.3483,E1 4.4757,E2 510.248} C_DIS
LIN {X 62.3081,Y -123.2037,Z 182,A -59.0215,B 4.3848,C 0.3493,E1 4.472,E2 511.7312} C_DIS
LIN {X 58.7325,Y -124.9503,Z 182,A -60.6057,B 4.3847,C 0.3507,E1 4.468,E2 513.3079} C_DIS
LIN {X 56.0831,Y -126.1591,Z 182,A -61.8011,B 4.3846,C 0.3521,E1 4.465,E2 514.5023} C_DIS
LIN {X 52.8713,Y -127.5386,Z 182,A -63.2243,B 4.3844,C 0.3536,E1 4.4613,E2 515.923} C_DIS
LIN {X 49.687,Y -128.8126,Z 182,A -64.6269,B 4.3844,C 0.355,E1 4.4577,E2 517.3239} C_DIS
LIN {X 46.489,Y -130.001,Z 182,A -66.0239,B 4.3842,C 0.3563,E1 4.454,E2 518.7194} C_DIS
LIN {X 43.2805,Y -131.1041,Z 182,A -67.428,B 4.3842,C 0.3577,E1 4.4503,E2 520.1239} C_DIS
LIN {X 39.5998,Y -132.2647,Z 182,A -68.9956,B 4.384,C 0.3589,E1 4.4461,E2 521.6882} C_DIS
LIN {X 36.3794,Y -133.1864,Z 182,A -70.3697,B 4.384,C 0.36,E1 4.4424,E2 523.061} C_DIS
LIN {X 33.6238,Y -133.9065,Z 182,A -71.5385,B 4.3839,C 0.3608,E1 4.4393,E2 524.2288} C_DIS
LIN {X 30.2781,Y -134.7029,Z 182,A -72.973,B 4.3838,C 0.362,E1 4.4354,E2 525.6651} C_DIS
LIN {X 26.7266,Y -135.4539,Z 182,A -74.4437,B 4.3838,C 0.3626,E1 4.4313,E2 527.1321} C_DIS
LIN {X 23.9842,Y -135.9643,Z 182,A -75.5903,B 4.3837,C 0.3633,E1 4.4282,E2 528.2779} C_DIS
LIN {X 20.7882,Y -136.4895,Z 182,A -76.9231,B 4.3836,C 0.3639,E1 4.4245,E2 529.61} C_DIS
LIN {X 17.6054,Y -136.9365,Z 182,A -78.2167,B 4.3836,C 0.3642,E1 4.4209,E2 530.8991} C_DIS
LIN {X 14.6187,Y -137.2872,Z 182,A -79.5102,B 4.3835,C 0.3652,E1 4.4173,E2 532.1992} C_DIS
LIN {X 10.835,Y -137.6397,Z 182,A -81.0539,B 4.3835,C 0.3655,E1 4.413,E2 533.7394} C_DIS
LIN {X 8.1602,Y -137.8223,Z 182,A -82.1598,B 4.3835,C 0.3658,E1 4.41,E2 534.8449} C_DIS
LIN {X 5.0541,Y -137.9712,Z 182,A -83.4811,B 4.3834,C 0.3664,E1 4.4063,E2 536.1709} C_DIS
LIN {X 0.9732,Y -138.06,Z 182,A -85.1818,B 4.3834,C 0.3668,E1 4.4015,E2 537.8734} C_DIS
Enddeposition()
LIN {X 0.9732,Y -138.06,Z 182,A -85.1818,B 4.3834,C 0.3668,E1 4.4015,E2 537.8734} C_DIS
Startdeposition()
$VEL.CP = VEL_PRINT
LIN {X 2.5964,Y -138.9409,Z 182,A -83.8442,B 4.3716,C 0.3619,E1 4.3933,E2 536.4819} C_DIS
LIN {X 5.6348,Y -138.8507,Z 182,A -82.5967,B 4.3716,C 0.3617,E1 4.3968,E2 535.2346} C_DIS
LIN {X 9.5681,Y -138.636,Z 182,A -80.8809,B 4.3718,C 0.3602,E1 4.4016,E2 533.5056} C_DIS
LIN {X 13.3284,Y -138.324,Z 182,A -79.4207,B 4.3718,C 0.3606,E1 4.4056,E2 532.0574} C_DIS
LIN {X 16.9848,Y -137.9238,Z 182,A -77.3239,B 4.3723,C 0.3536,E1 4.4117,E2 529.8816} C_DIS
LIN {X 21.956,Y -137.2209,Z 182,A -75.882,B 4.3718,C 0.3593,E1 4.4154,E2 528.5232} C_DIS
LIN {X 26.2601,Y -136.4609,Z 182,A -74.0732,B 4.3719,C 0.3581,E1 4.4204,E2 526.7124} C_DIS
LIN {X 30.0569,Y -135.6771,Z 182,A -71.9663,B 4.3725,C 0.3513,E1 4.4263,E2 524.5361} C_DIS
LIN {X 34.4008,Y -134.6394,Z 182,A -70.6255,B 4.3722,C 0.3553,E1 4.4298,E2 523.2616} C_DIS
LIN {X 37.7833,Y -133.7299,Z 182,A -69.1962,B 4.3722,C 0.3542,E1 4.4336,E2 521.8334} C_DIS
LIN {X 41.1453,Y -132.7344,Z 182,A -67.8275,B 4.3722,C 0.3537,E1 4.4373,E2 520.474} C_DIS
LIN {X 44.1414,Y -131.7676,Z 182,A -66.494,B 4.3724,C 0.352,E1 4.4408,E2 519.1348} C_DIS
LIN {X 47.9928,Y -130.4163,Z 182,A -64.8733,B 4.3725,C 0.3509,E1 4.445,E2 517.5214} C_DIS
LIN {X 50.6759,Y -129.3953,Z 182,A -63.6785,B 4.3726,C 0.3494,E1 4.4482,E2 516.3242} C_DIS
LIN {X 53.788,Y -128.1327,Z 182,A -62.3063,B 4.3728,C 0.3479,E1 4.4517,E2 514.9527} C_DIS
LIN {X 56.9538,Y -126.7572,Z 182,A -60.9252,B 4.3728,C 0.3466,E1 4.4552,E2 513.5762} C_DIS
LIN {X 60.1599,Y -125.2674,Z 182,A -59.4303,B 4.373,C 0.3442,E1 4.459,E2 512.0752} C_DIS
LIN {X 63.7443,Y -123.4841,Z 182,A -57.857,B 4.3732,C 0.3428,E1 4.4629,E2 510.5111} C_DIS
LIN {X 66.7592,Y -121.8806,Z 182,A -56.2065,B 4.3735,C 0.3379,E1 4.467,E2 508.827} C_DIS
LIN {X 72.1921,Y -118.7435,Z 182,A -53.8283,B 4.3737,C 0.3364,E1 4.4727,E2 506.4748} C_DIS
LIN {X 76.035,Y -116.3206,Z 182,A -51.9643,B 4.3739,C 0.3335,E1 4.4771,E2 504.6105} C_DIS
LIN {X 79.7735,Y -113.7891,Z 182,A -49.9502,B 4.3743,C 0.3284,E1 4.4818,E2 502.5746} C_DIS
LIN {X 82.6051,Y -111.7505,Z 182,A -49.009,B 4.374,C 0.3319,E1 4.4837,E2 501.6988} C_DIS
LIN {X 86.4571,Y -108.7971,Z 182,A -46.811,B 4.3744,C 0.3259,E1 4.4887,E2 499.4729} C_DIS
LIN {X 89.9794,Y -105.9024,Z 182,A -45.1556,B 4.3745,C 0.3251,E1 4.4921,E2 497.8459} C_DIS
LIN {X 92.5156,Y -103.6945,Z 182,A -43.5977,B 4.3749,C 0.3202,E1 4.4955,E2 496.264} C_DIS
LIN {X 95.8814,Y -100.5903,Z 182,A -41.7567,B 4.3751,C 0.317,E1 4.4992,E2 494.4277} C_DIS
LIN {X 99.1038,Y -97.4171,Z 182,A -39.9286,B 4.3753,C 0.3136,E1 4.5028,E2 492.6028} C_DIS
LIN {X 105.6316,Y -90.2971,Z 182,A -36.116,B 4.3758,C 0.3071,E1 4.5099,E2 488.8098} C_DIS
LIN {X 107.7411,Y -87.7697,Z 182,A -34.4046,B 4.3763,C 0.2995,E1 4.513,E2 487.05} C_DIS
LIN {X 110.276,Y -84.5628,Z 182,A -33.089,B 4.3763,C 0.3004,E1 4.5152,E2 485.7824} C_DIS
LIN {X 112.9867,Y -80.9051,Z 182,A -31.28,B 4.3765,C 0.2968,E1 4.5181,E2 483.9808} C_DIS
LIN {X 115.5256,Y -77.2364,Z 182,A -29.4743,B 4.3768,C 0.2928,E1 4.521,E2 482.1781} C_DIS
LIN {X 118.2421,Y -73.0109,Z 182,A -27.6447,B 4.3769,C 0.2909,E1 4.5236,E2 480.3786} C_DIS
LIN {X 119.8832,Y -70.2827,Z 182,A -26.2002,B 4.3772,C 0.2859,E1 4.5257,E2 478.9156} C_DIS
LIN {X 122.1601,Y -66.2469,Z 182,A -24.3151,B 4.3775,C 0.2814,E1 4.5283,E2 477.0323} C_DIS
LIN {X 124.0313,Y -62.6696,Z 182,A -22.7578,B 4.3777,C 0.2786,E1 4.5302,E2 475.4877} C_DIS
LIN {X 125.5832,Y -59.499,Z 182,A -21.4004,B 4.3779,C 0.2761,E1 4.5319,E2 474.142} C_DIS
LIN {X 126.9572,Y -56.5066,Z 182,A -20.0565,B 4.3781,C 0.2727,E1 4.5334,E2 472.7987} C_DIS
LIN {X 128.3555,Y -53.2545,Z 182,A -18.6357,B 4.3783,C 0.2693,E1 4.535,E2 471.3818} C_DIS
LIN {X 129.6557,Y -50.0061,Z 182,A -17.2172,B 4.3785,C 0.2658,E1 4.5364,E2 469.9653} C_DIS
LIN {X 130.8472,Y -46.7999,Z 182,A -15.8761,B 4.3787,C 0.2629,E1 4.5377,E2 468.6322} C_DIS
LIN {X 131.9583,Y -43.5688,Z 182,A -14.5027,B 4.3789,C 0.2596,E1 4.5389,E2 467.2623} C_DIS
LIN {X 133.3664,Y -39.0451,Z 182,A -12.4802,B 4.3792,C 0.2533,E1 4.5405,E2 465.229} C_DIS
LIN {X 134.7631,Y -33.9133,Z 182,A -10.5072,B 4.3794,C 0.2501,E1 4.5419,E2 463.2832} C_DIS
LIN {X 135.4626,Y -31.0001,Z 182,A -9.275,B 4.3796,C 0.2468,E1 4.5427,E2 462.0504} C_DIS
LIN {X 136.2571,Y -27.3004,Z 182,A -7.7363,B 4.3798,C 0.2427,E1 4.5436,E2 460.5133} C_DIS
LIN {X 137.0265,Y -23.1291,Z 182,A -5.7737,B 4.3803,C 0.235,E1 4.5445,E2 458.5213} C_DIS
LIN {X 137.5711,Y -19.6303,Z 182,A -4.6813,B 4.3803,C 0.2357,E1 4.5449,E2 457.4759} C_DIS
LIN {X 138.036,Y -16.0439,Z 182,A -3.1133,B 4.3805,C 0.2305,E1 4.5455,E2 455.8968} C_DIS
LIN {X 138.4747,Y -11.6594,Z 182,A -1.4563,B 4.3807,C 0.2274,E1 4.5459,E2 454.2593} C_DIS
LIN {X 138.7578,Y -7.6087,Z 182,A 0.1738,B 4.3809,C 0.2233,E1 4.5462,E2 452.6337} C_DIS
LIN {X 138.9079,Y -3.9773,Z 182,A 1.6782,B 4.3811,C 0.2189,E1 4.5463,E2 451.1275} C_DIS
LIN {X 138.9649,Y 0.5402,Z 182,A 3.4731,B 4.3813,C 0.2146,E1 4.5463,E2 449.3401} C_DIS
LIN {X 138.889,Y 4.6531,Z 182,A 5.1709,B 4.3815,C 0.2097,E1 4.5463,E2 447.6409} C_DIS
LIN {X 138.6899,Y 8.738,Z 182,A 6.6675,B 4.3816,C 0.2074,E1 4.546,E2 446.1677} C_DIS
LIN {X 138.3682,Y 12.869,Z 182,A 8.8486,B 4.3822,C 0.1964,E1 4.5454,E2 443.9239} C_DIS
LIN {X 137.8536,Y 17.5447,Z 182,A 11.0831,B 4.3826,C 0.1871,E1 4.5446,E2 441.6495} C_DIS
LIN {X 136.8502,Y 24.1514,Z 182,A 12.6891,B 4.3822,C 0.1944,E1 4.5439,E2 440.1915} C_DIS
LIN {X 135.9351,Y 28.862,Z 182,A 14.6556,B 4.3825,C 0.1891,E1 4.5429,E2 438.2254} C_DIS
LIN {X 135.287,Y 31.768,Z 182,A 15.9654,B 4.3827,C 0.1846,E1 4.542,E2 436.9044} C_DIS
LIN {X 134.6112,Y 34.5119,Z 182,A 17.047,B 4.3827,C 0.1825,E1 4.5413,E2 435.8328} C_DIS
LIN {X 133.8535,Y 37.3411,Z 182,A 18.2729,B 4.3829,C 0.1789,E1 4.5404,E2 434.6039} C_DIS
LIN {X 132.8767,Y 40.6803,Z 182,A 19.7066,B 4.3831,C 0.175,E1 4.5393,E2 433.1694} C_DIS
LIN {X 131.7657,Y 44.1472,Z 182,A 21.1425,B 4.3831,C 0.1718,E1 4.538,E2 431.7411} C_DIS
LIN {X 130.3748,Y 48.1037,Z 182,A 23.8793,B 4.3838,C 0.1543,E1 4.5353,E2 428.8728} C_DIS
LIN {X 127.4905,Y 55.2925,Z 182,A 25.9611,B 4.3836,C 0.1602,E1 4.5331,E2 426.9337} C_DIS
LIN {X 125.4461,Y 59.7859,Z 182,A 27.6894,B 4.3836,C 0.1588,E1 4.5311,E2 425.2438} C_DIS
LIN {X 124.3481,Y 62.0402,Z 182,A 28.8942,B 4.3838,C 0.154,E1 4.5296,E2 424.0167} C_DIS
LIN {X 122.551,Y 65.5208,Z 182,A 30.567,B 4.384,C 0.1492,E1 4.5274,E2 422.336} C_DIS
LIN {X 118.1281,Y 73.1946,Z 182,A 33.9527,B 4.3842,C 0.1436,E1 4.5227,E2 418.983} C_DIS
LIN {X 116.7031,Y 75.4458,Z 182,A 35.1917,B 4.3843,C 0.1392,E1 4.5208,E2 417.7257} C_DIS
LIN {X 114.153,Y 79.2511,Z 182,A 36.9959,B 4.3844,C 0.1358,E1 4.518,E2 415.9317} C_DIS
LIN {X 111.5657,Y 82.8538,Z 182,A 38.8006,B 4.3846,C 0.1319,E1 4.515,E2 414.1295} C_DIS
LIN {X 108.7144,Y 86.561,Z 182,A 40.7438,B 4.3846,C 0.1274,E1 4.5117,E2 412.1838} C_DIS
LIN {X 105.6434,Y 90.2841,Z 182,A 42.5839,B 4.3848,C 0.1249,E1 4.5084,E2 410.3624} C_DIS
LIN {X 102.7048,Y 93.6133,Z 182,A 44.3921,B 4.3848,C 0.1212,E1 4.505,E2 408.5566} C_DIS
LIN {X 99.6845,Y 96.8228,Z 182,A 46.1637,B 4.385,C 0.118,E1 4.5016,E2 406.7904} C_DIS
LIN {X 95.8467,Y 100.6235,Z 182,A 48.0698,B 4.385,C 0.1174,E1 4.4979,E2 404.9245} C_DIS
LIN {X 92.9322,Y 103.3214,Z 182,A 49.9799,B 4.3851,C 0.1109,E1 4.4939,E2 402.9797} C_DIS
LIN {X 89.6089,Y 106.2168,Z 182,A 51.7109,B 4.3852,C 0.1086,E1 4.4902,E2 401.2594} C_DIS
LIN {X 86.7677,Y 108.5499,Z 182,A 53.2329,B 4.3852,C 0.1057,E1 4.4869,E2 399.7365} C_DIS
LIN {X 83.2998,Y 111.2336,Z 182,A 55.0081,B 4.3853,C 0.1029,E1 4.483,E2 397.9653} C_DIS
LIN {X 76.9836,Y 115.6944,Z 182,A 58.1476,B 4.3854,C 0.0982,E1 4.4758,E2 394.8319} C_DIS
LIN {X 73.0109,Y 118.2421,Z 182,A 59.9401,B 4.3854,C 0.0969,E1 4.4716,E2 393.0587} C_DIS
LIN {X 69.675,Y 120.2373,Z 182,A 61.5685,B 4.3855,C 0.0943,E1 4.4677,E2 391.4271} C_DIS
LIN {X 65.9242,Y 122.3342,Z 182,A 63.4077,B 4.3856,C 0.091,E1 4.4631,E2 389.5795} C_DIS
LIN {X 62.0289,Y 124.3537,Z 182,A 65.7382,B 4.3858,C 0.0828,E1 4.4572,E2 387.1832} C_DIS
LIN {X 56.9682,Y 126.7508,Z 182,A 67.1749,B 4.3856,C 0.0896,E1 4.4538,E2 385.8567} C_DIS
LIN {X 53.1116,Y 128.4152,Z 182,A 68.9801,B 4.3856,C 0.0868,E1 4.4491,E2 384.0426} C_DIS
LIN {X 50.0609,Y 129.6344,Z 182,A 70.3726,B 4.3857,C 0.0849,E1 4.4455,E2 382.6456} C_DIS
LIN {X 46.1753,Y 131.0703,Z 182,A 72.3279,B 4.3858,C 0.0805,E1 4.4402,E2 380.6596} C_DIS
LIN {X 43.0109,Y 132.1429,Z 182,A 73.367,B 4.3858,C 0.0828,E1 4.4376,E2 379.6632} C_DIS
LIN {X 40.3167,Y 132.988,Z 182,A 74.4902,B 4.3858,C 0.0822,E1 4.4346,E2 378.5453} C_DIS
LIN {X 36.9073,Y 133.9748,Z 182,A 75.9846,B 4.3858,C 0.0807,E1 4.4306,E2 377.0474} C_DIS
LIN {X 33.7373,Y 134.8078,Z 182,A 77.462,B 4.3858,C 0.0783,E1 4.4265,E2 375.5546} C_DIS
LIN {X 26.449,Y 136.4248,Z 182,A 80.5572,B 4.3858,C 0.0761,E1 4.4181,E2 372.4581} C_DIS
LIN {X 17.6625,Y 137.8382,Z 182,A 84.0225,B 4.3858,C 0.0764,E1 4.4086,E2 369.0197} C_DIS
LIN {X 13.8051,Y 138.2783,Z 182,A 85.7234,B 4.3859,C 0.0748,E1 4.4038,E2 367.3069} C_DIS
LIN {X 10.0274,Y 138.6025,Z 182,A 87.2149,B 4.3859,C 0.0751,E1 4.3997,E2 365.825} C_DIS
LIN {X 6.6824,Y 138.8043,Z 182,A 88.6554,B 4.3859,C 0.0742,E1 4.3957,E2 364.3776} C_DIS
LIN {X 2.3801,Y 138.9445,Z 182,A 90.359,B 4.3859,C 0.0746,E1 4.3909,E2 362.6837} C_DIS
LIN {X -1.7013,Y 138.9558,Z 182,A 92.1322,B 4.3859,C 0.0737,E1 4.3859,E2 360.8999} C_DIS
LIN {X -5.5003,Y 138.8559,Z 182,A 93.6335,B 4.3859,C 0.0743,E1 4.3818,E2 359.4075} C_DIS
LIN {X -9.9709,Y 138.6066,Z 182,A 96.0656,B 4.386,C 0.069,E1 4.3748,E2 356.9029} C_DIS
LIN {X -15.0344,Y 138.1491,Z 182,A 97.532,B 4.3859,C 0.0754,E1 4.3709,E2 355.5164} C_DIS
LIN {X -18.6617,Y 137.7072,Z 182,A 99.4847,B 4.3859,C 0.0717,E1 4.3654,E2 353.5088} C_DIS
LIN {X -22.5669,Y 137.1203,Z 182,A 100.493,B 4.3859,C 0.078,E1 4.3628,E2 352.5788} C_DIS
LIN {X -26.3182,Y 136.4498,Z 182,A 102.3173,B 4.3859,C 0.0764,E1 4.3577,E2 350.7239} C_DIS
LIN {X -29.5681,Y 135.7826,Z 182,A 103.6764,B 4.3859,C 0.0772,E1 4.354,E2 349.3667} C_DIS
LIN {X -32.9421,Y 135.0041,Z 182,A 105.1899,B 4.3859,C 0.0773,E1 4.3499,E2 347.8433} C_DIS
LIN {X -37.9615,Y 133.68,Z 182,A 107.1855,B 4.3859,C 0.08,E1 4.3445,E2 345.867} C_DIS
LIN {X -40.8612,Y 132.8213,Z 182,A 108.5032,B 4.3859,C 0.0804,E1 4.341,E2 344.5412} C_DIS
LIN {X -44.2426,Y 131.7339,Z 182,A 109.9833,B 4.3858,C 0.0814,E1 4.3371,E2 343.0602} C_DIS
LIN {X -47.6535,Y 130.5394,Z 182,A 111.4921,B 4.3858,C 0.0826,E1 4.3331,E2 341.55} C_DIS
LIN {X -56.5104,Y 126.9555,Z 182,A 115.2513,B 4.3857,C 0.0882,E1 4.3235,E2 337.8161} C_DIS
LIN {X -60.8066,Y 124.9567,Z 182,A 117.4168,B 4.3857,C 0.0887,E1 4.3179,E2 335.6258} C_DIS
LIN {X -63.4333,Y 123.6425,Z 182,A 118.6971,B 4.3857,C 0.0896,E1 4.3147,E2 334.3376} C_DIS
LIN {X -66.7649,Y 121.8775,Z 182,A 120.3549,B 4.3857,C 0.0908,E1 4.3106,E2 332.6681} C_DIS
LIN {X -70.7632,Y 119.6008,Z 182,A 122.241,B 4.3856,C 0.0935,E1 4.306,E2 330.7847} C_DIS
LIN {X -74.4422,Y 117.346,Z 182,A 124.1019,B 4.3856,C 0.0954,E1 4.3016,E2 328.9149} C_DIS
LIN {X -78.2346,Y 114.8527,Z 182,A 126.0293,B 4.3855,C 0.0978,E1 4.2971,E2 326.9819} C_DIS
LIN {X -82.4237,Y 111.8838,Z 182,A 128.1008,B 4.3854,C 0.1016,E1 4.2924,E2 324.9177} C_DIS
LIN {X -85.2725,Y 109.728,Z 182,A 129.6791,B 4.3854,C 0.1033,E1 4.2889,E2 323.3274} C_DIS
LIN {X -88.8786,Y 106.8285,Z 182,A 131.6091,B 4.3853,C 0.1065,E1 4.2847,E2 321.396} C_DIS
LIN {X -92.7536,Y 103.4813,Z 182,A 133.9092,B 4.3852,C 0.1089,E1 4.2799,E2 319.0739} C_DIS
LIN {X -95.6663,Y 100.7956,Z 182,A 135.4485,B 4.3851,C 0.1127,E1 4.2768,E2 317.5479} C_DIS
LIN {X -98.9211,Y 97.6033,Z 182,A 137.3645,B 4.3851,C 0.1162,E1 4.273,E2 315.6287} C_DIS
LIN {X -102.4315,Y 93.9118,Z 182,A 139.4445,B 4.3849,C 0.1206,E1 4.269,E2 313.553} C_DIS
LIN {X -104.2476,Y 91.8918,Z 182,A 140.6117,B 4.3849,C 0.1226,E1 4.2668,E2 312.3807} C_DIS
LIN {X -107.1058,Y 88.5437,Z 182,A 142.5028,B 4.3847,C 0.126,E1 4.2634,E2 310.4816} C_DIS
LIN {X -109.9483,Y 84.9883,Z 182,A 144.5333,B 4.3847,C 0.129,E1 4.2599,E2 308.4333} C_DIS
LIN {X -112.8138,Y 81.147,Z 182,A 146.4784,B 4.3845,C 0.1337,E1 4.2567,E2 306.4937} C_DIS
LIN {X -115.3461,Y 77.5053,Z 182,A 148.4029,B 4.3845,C 0.1373,E1 4.2536,E2 304.5587} C_DIS
LIN {X -117.8019,Y 73.7187,Z 182,A 150.2169,B 4.3842,C 0.142,E1 4.2509,E2 302.7521} C_DIS
LIN {X -119.821,Y 70.3886,Z 182,A 151.9248,B 4.3842,C 0.1452,E1 4.2485,E2 301.0326} C_DIS
LIN {X -122.1149,Y 66.3297,Z 182,A 154.369,B 4.3842,C 0.1463,E1 4.2451,E2 298.5237} C_DIS
LIN {X -124.2782,Y 62.1819,Z 182,A 155.7683,B 4.3838,C 0.1549,E1 4.2434,E2 297.1933} C_DIS
LIN {X -125.4494,Y 59.7789,Z 182,A 156.9991,B 4.3838,C 0.1568,E1 4.2419,E2 295.947} C_DIS
LIN {X -126.8773,Y 56.6852,Z 182,A 158.3383,B 4.3836,C 0.1609,E1 4.2404,E2 294.6173} C_DIS
LIN {X -128.1418,Y 53.7662,Z 182,A 160.2528,B 4.3836,C 0.1602,E1 4.2382,E2 292.6271} C_DIS
LIN {X -129.8349,Y 49.5421,Z 182,A 161.6233,B 4.3833,C 0.1686,E1 4.2369,E2 291.3228} C_DIS
LIN {X -131.0973,Y 46.0974,Z 182,A 163.1366,B 4.3832,C 0.1726,E1 4.2355,E2 289.8106} C_DIS
LIN {X -132.3672,Y 42.3087,Z 182,A 164.9341,B 4.383,C 0.176,E1 4.2339,E2 287.9954} C_DIS
LIN {X -133.3812,Y 38.9945,Z 182,A 166.381,B 4.3829,C 0.1798,E1 4.2327,E2 286.5473} C_DIS
LIN {X -134.2752,Y 35.7952,Z 182,A 167.8947,B 4.3828,C 0.1826,E1 4.2316,E2 285.0163} C_DIS
LIN {X -135.1558,Y 32.3126,Z 182,A 169.3521,B 4.3826,C 0.1868,E1 4.2307,E2 283.5632} C_DIS
LIN {X -135.9028,Y 29.0116,Z 182,A 170.9613,B 4.3825,C 0.1892,E1 4.2297,E2 281.9277} C_DIS
LIN {X -136.7986,Y 24.4396,Z 182,A 172.7975,B 4.3822,C 0.1952,E1 4.2287,E2 280.1039} C_DIS
LIN {X -137.3971,Y 20.8183,Z 182,A 174.3033,B 4.382,C 0.1995,E1 4.2281,E2 278.6003} C_DIS
LIN {X -137.8375,Y 17.6678,Z 182,A 175.6984,B 4.3819,C 0.2026,E1 4.2276,E2 277.1954} C_DIS
LIN {X -138.3783,Y 12.7633,Z 182,A 178.1196,B 4.3817,C 0.2057,E1 4.2269,E2 274.7261} C_DIS
LIN {X -138.6542,Y 9.3131,Z 182,A 179.2342,B 4.3814,C 0.2119,E1 4.2267,E2 273.6527} C_DIS
LIN {X -138.8039,Y 6.691,Z 182,A -179.6172,B 4.3814,C 0.2145,E1 4.2265,E2 272.4965} C_DIS
LIN {X -138.9313,Y 3.1376,Z 182,A -177.613,B 4.3813,C 0.215,E1 4.2264,E2 270.424} C_DIS
LIN {X -138.962,Y -1.0037,Z 182,A -176.1061,B 4.381,C 0.2212,E1 4.2264,E2 268.9442} C_DIS
LIN {X -138.8652,Y -5.2615,Z 182,A -174.4591,B 4.3807,C 0.2269,E1 4.2265,E2 267.3125} C_DIS
LIN {X -138.6696,Y -9.0677,Z 182,A -172.749,B 4.3805,C 0.2304,E1 4.2268,E2 265.5856} C_DIS
LIN {X -138.2283,Y -14.2986,Z 182,A -170.5508,B 4.3802,C 0.2363,E1 4.2274,E2 263.3845} C_DIS
LIN {X -137.7213,Y -18.5544,Z 182,A -168.8391,B 4.3799,C 0.2416,E1 4.228,E2 261.6812} C_DIS
LIN {X -137.2832,Y -21.5538,Z 182,A -167.5315,B 4.3797,C 0.2447,E1 4.2285,E2 260.3668} C_DIS
LIN {X -136.7321,Y -24.811,Z 182,A -166.1661,B 4.3795,C 0.2485,E1 4.2292,E2 259.0018} C_DIS
LIN {X -136.1664,Y -27.7464,Z 182,A -164.8277,B 4.3794,C 0.2512,E1 4.2299,E2 257.6505} C_DIS
LIN {X -135.4736,Y -30.9522,Z 182,A -163.4371,B 4.3792,C 0.2547,E1 4.2308,E2 256.2556} C_DIS
LIN {X -134.6546,Y -34.3409,Z 182,A -161.9526,B 4.379,C 0.2583,E1 4.2318,E2 254.7659} C_DIS
LIN {X -133.7281,Y -37.7895,Z 182,A -160.4067,B 4.3787,C 0.2617,E1 4.2329,E2 253.2113} C_DIS
LIN {X -132.7984,Y -40.9363,Z 182,A -159.0124,B 4.3785,C 0.2651,E1 4.2341,E2 251.8123} C_DIS
LIN {X -131.5195,Y -44.8796,Z 182,A -156.8923,B 4.3785,C 0.2668,E1 4.236,E2 249.6395} C_DIS
LIN {X -130.2822,Y -48.3509,Z 182,A -155.8767,B 4.378,C 0.2743,E1 4.2369,E2 248.6905} C_DIS
LIN {X -128.7007,Y -52.4161,Z 182,A -153.873,B 4.3778,C 0.2776,E1 4.239,E2 246.661} C_DIS
LIN {X -127.4574,Y -55.3691,Z 182,A -152.4465,B 4.3776,C 0.2802,E1 4.2406,E2 245.2213} C_DIS
LIN {X -126.0041,Y -58.6015,Z 182,A -150.9792,B 4.3774,C 0.2839,E1 4.2423,E2 243.7539} C_DIS
LIN {X -124.4105,Y -61.9137,Z 182,A -149.2897,B 4.3772,C 0.2864,E1 4.2444,E2 242.0422} C_DIS
LIN {X -121.2095,Y -67.9698,Z 182,A -146.7521,B 4.3766,C 0.2955,E1 4.2477,E2 239.5435} C_DIS
LIN {X -118.7693,Y -72.1495,Z 182,A -144.4036,B 4.3765,C 0.2977,E1 4.2511,E2 237.1495} C_DIS
LIN {X -116.3982,Y -75.9156,Z 182,A -142.4858,B 4.3762,C 0.3013,E1 4.254,E2 235.2215} C_DIS
LIN {X -113.9697,Y -79.5145,Z 182,A -140.651,B 4.3759,C 0.3051,E1 4.2569,E2 233.3814} C_DIS
LIN {X -110.7585,Y -83.9296,Z 182,A -138.4285,B 4.3756,C 0.3103,E1 4.2606,E2 231.1634} C_DIS
LIN {X -108.3003,Y -87.0788,Z 182,A -136.6201,B 4.3754,C 0.3126,E1 4.2638,E2 229.3341} C_DIS
LIN {X -105.5143,Y -90.4348,Z 182,A -134.7858,B 4.3752,C 0.3161,E1 4.2671,E2 227.4956} C_DIS
LIN {X -102.6038,Y -93.7244,Z 182,A -132.9729,B 4.3749,C 0.3198,E1 4.2705,E2 225.6828} C_DIS
LIN {X -99.595,Y -96.9153,Z 182,A -131.0921,B 4.3747,C 0.3228,E1 4.2741,E2 223.7928} C_DIS
LIN {X -96.3278,Y -100.1637,Z 182,A -129.1403,B 4.3744,C 0.326,E1 4.278,E2 221.8344} C_DIS
LIN {X -93.1212,Y -103.1513,Z 182,A -127.332,B 4.3742,C 0.3293,E1 4.2817,E2 220.0262} C_DIS
LIN {X -89.7599,Y -106.0891,Z 182,A -125.4302,B 4.374,C 0.332,E1 4.2858,E2 218.1165} C_DIS
LIN {X -86.2489,Y -108.9628,Z 182,A -123.5241,B 4.3738,C 0.3348,E1 4.29,E2 216.2058} C_DIS
LIN {X -77.8473,Y -115.1148,Z 182,A -119.3992,B 4.3731,C 0.343,E1 4.2993,E2 212.1038} C_DIS
LIN {X -74.6857,Y -117.1911,Z 182,A -117.7902,B 4.373,C 0.3448,E1 4.303,E2 210.4883} C_DIS
LIN {X -71.9061,Y -118.9165,Z 182,A -116.2081,B 4.373,C 0.3447,E1 4.3069,E2 208.8752} C_DIS
LIN {X -67.967,Y -121.2111,Z 182,A -114.2776,B 4.3729,C 0.3467,E1 4.3116,E2 206.9379} C_DIS
LIN {X -64.3334,Y -123.1761,Z 182,A -111.9161,B 4.3731,C 0.3429,E1 4.3176,E2 204.4878} C_DIS
LIN {X -59.1345,Y -125.7573,Z 182,A -109.9071,B 4.3727,C 0.349,E1 4.3226,E2 202.5304} C_DIS
LIN {X -56.0348,Y -127.1682,Z 182,A -108.6489,B 4.3724,C 0.3517,E1 4.3257,E2 201.2915} C_DIS
LIN {X -52.012,Y -128.8636,Z 182,A -106.9605,B 4.3722,C 0.3545,E1 4.3301,E2 199.6177} C_DIS
LIN {X -48.734,Y -130.1387,Z 182,A -105.2569,B 4.3723,C 0.3534,E1 4.3346,E2 197.8799} C_DIS
LIN {X -43.7791,Y -131.8882,Z 182,A -103.3503,B 4.372,C 0.3576,E1 4.3396,E2 196.0077} C_DIS
LIN {X -39.978,Y -133.0916,Z 182,A -101.689,B 4.3719,C 0.3586,E1 4.344,E2 194.3438} C_DIS
LIN {X -36.2528,Y -134.1531,Z 182,A -99.9739,B 4.3719,C 0.3584,E1 4.3486,E2 192.6124} C_DIS
LIN {X -29.0821,Y -135.8876,Z 182,A -97.2458,B 4.3715,C 0.363,E1 4.356,E2 189.9255} C_DIS
LIN {X -26.7088,Y -136.3751,Z 182,A -95.769,B 4.3719,C 0.3588,E1 4.3602,E2 188.3845} C_DIS
LIN {X -22.7824,Y -137.0844,Z 182,A -94.2848,B 4.3717,C 0.361,E1 4.3642,E2 186.9212} C_DIS
LIN {X -19.2184,Y -137.63,Z 182,A -92.8053,B 4.3717,C 0.3614,E1 4.3683,E2 185.4422} C_DIS
LIN {X -15.098,Y -138.1423,Z 182,A -91.1226,B 4.3717,C 0.3621,E1 4.373,E2 183.7627} C_DIS
LIN {X -11.5396,Y -138.4849,Z 182,A -89.6297,B 4.3717,C 0.3621,E1 4.3771,E2 182.2667} C_DIS
LIN {X -6.9963,Y -138.7885,Z 182,A -87.7572,B 4.3716,C 0.3621,E1 4.3823,E2 180.3941} C_DIS
LIN {X -3.2895,Y -138.927,Z 182,A -86.1386,B 4.3716,C 0.3611,E1 4.3869,E2 178.7628} C_DIS
LIN {X 0.9838,Y -138.96,Z 182,A -84.5716,B 4.3716,C 0.3629,E1 4.3912,E2 177.221} C_DIS
Enddeposition()
LIN {X 0.9838,Y -138.96,Z 182,A -84.5716,B 4.3716,C 0.3629,E1 4.3912,E2 177.221} C_DIS
Startdeposition()
$VEL.CP = VEL_PRINT
LIN {X -1.4047,Y -139.8607,Z 182,A -86.1819,B 4.3579,C 0.3717,E1 4.3735,E2 178.9519} C_DIS
LIN {X -5.4218,Y -139.7611,Z 182,A -87.7711,B 4.3579,C 0.3711,E1 4.3691,E2 180.5342} C_DIS
LIN {X -9.5191,Y -139.5435,Z 182,A -89.5012,B 4.3579,C 0.3716,E1 4.3642,E2 182.2717} C_DIS
LIN {X -13.4237,Y -139.2205,Z 182,A -91.0247,B 4.3579,C 0.3706,E1 4.36,E2 183.7849} C_DIS
LIN {X -17.6838,Y -138.7446,Z 182,A -92.8599,B 4.3579,C 0.371,E1 4.3549,E2 185.6314} C_DIS
LIN {X -21.9516,Y -138.1338,Z 182,A -94.5411,B 4.358,C 0.3697,E1 4.3503,E2 187.3018} C_DIS
LIN {X -26.4611,Y -137.3403,Z 182,A -96.4561,B 4.358,C 0.3694,E1 4.345,E2 189.2227} C_DIS
LIN {X -30.7025,Y -136.4553,Z 182,A -98.3751,B 4.358,C 0.3699,E1 4.3397,E2 191.1615} C_DIS
LIN {X -37.7189,Y -134.6839,Z 182,A -101.1684,B 4.3583,C 0.3666,E1 4.3322,E2 193.9328} C_DIS
LIN {X -40.8925,Y -133.7545,Z 182,A -102.536,B 4.3583,C 0.3658,E1 4.3285,E2 195.3024} C_DIS
LIN {X -43.9625,Y -132.7773,Z 182,A -104.6102,B 4.3579,C 0.3717,E1 4.3228,E2 197.477} C_DIS
LIN {X -49.354,Y -130.8691,Z 182,A -106.2903,B 4.3585,C 0.3637,E1 4.3186,E2 199.0698} C_DIS
LIN {X -53.4709,Y -129.2421,Z 182,A -108.0868,B 4.3587,C 0.3618,E1 4.3139,E2 200.8643} C_DIS
LIN {X -56.7112,Y -127.8533,Z 182,A -109.6369,B 4.3587,C 0.3613,E1 4.3099,E2 202.4288} C_DIS
LIN {X -60.1542,Y -126.2692,Z 182,A -110.8945,B 4.3591,C 0.357,E1 4.3068,E2 203.6472} C_DIS
LIN {X -64.8072,Y -123.9456,Z 182,A -113.2705,B 4.3591,C 0.3567,E1 4.3008,E2 206.0561} C_DIS
LIN {X -69.0985,Y -121.6077,Z 182,A -115.4233,B 4.3592,C 0.3555,E1 4.2955,E2 208.2292} C_DIS
LIN {X -73.1095,Y -119.2392,Z 182,A -117.2864,B 4.3594,C 0.3525,E1 4.2911,E2 210.0864} C_DIS
LIN {X -76.7009,Y -116.9616,Z 182,A -119.1327,B 4.3596,C 0.3509,E1 4.2867,E2 211.9465} C_DIS
LIN {X -79.4762,Y -115.0942,Z 182,A -120.8718,B 4.3595,C 0.3519,E1 4.2826,E2 213.7343} C_DIS
LIN {X -82.8678,Y -112.6758,Z 182,A -122.4488,B 4.3598,C 0.3482,E1 4.2791,E2 215.2941} C_DIS
LIN {X -85.5675,Y -110.64,Z 182,A -123.6634,B 4.3601,C 0.3445,E1 4.2764,E2 216.4862} C_DIS
LIN {X -89.2243,Y -107.7126,Z 182,A -125.5774,B 4.3603,C 0.3412,E1 4.2723,E2 218.3993} C_DIS
LIN {X -92.5004,Y -104.9128,Z 182,A -127.4063,B 4.3606,C 0.3386,E1 4.2684,E2 220.2363} C_DIS
LIN {X -95.7296,Y -101.9752,Z 182,A -129.2725,B 4.3608,C 0.3359,E1 4.2646,E2 222.1127} C_DIS
LIN {X -98.8216,Y -98.9818,Z 182,A -131.0271,B 4.361,C 0.3325,E1 4.2611,E2 223.8659} C_DIS
LIN {X -101.8259,Y -95.8879,Z 182,A -132.8207,B 4.3613,C 0.3292,E1 4.2576,E2 225.6626} C_DIS
LIN {X -104.7879,Y -92.6416,Z 182,A -134.6988,B 4.3615,C 0.3262,E1 4.2541,E2 227.5505} C_DIS
LIN {X -107.7596,Y -89.1675,Z 182,A -136.5954,B 4.3618,C 0.3224,E1 4.2507,E2 229.4498} C_DIS
LIN {X -110.5945,Y -85.6262,Z 182,A -138.3751,B 4.3621,C 0.3178,E1 4.2476,E2 231.2187} C_DIS
LIN {X -112.5583,Y -83.0281,Z 182,A -139.9129,B 4.3622,C 0.3164,E1 4.245,E2 232.7828} C_DIS
LIN {X -115.2196,Y -79.2934,Z 182,A -141.83,B 4.3625,C 0.3124,E1 4.2419,E2 234.7043} C_DIS
LIN {X -117.0971,Y -76.4946,Z 182,A -143.3939,B 4.3626,C 0.3106,E1 4.2395,E2 236.2917} C_DIS
LIN {X -120.1526,Y -71.5985,Z 182,A -146.6644,B 4.3626,C 0.3115,E1 4.2346,E2 239.6787} C_DIS
LIN {X -123.7953,Y -65.0932,Z 182,A -148.7092,B 4.3636,C 0.2968,E1 4.2321,E2 241.5914} C_DIS
LIN {X -125.38,Y -61.9861,Z 182,A -150.1749,B 4.3638,C 0.2935,E1 4.2302,E2 243.0614} C_DIS
LIN {X -126.8477,Y -58.9249,Z 182,A -151.8434,B 4.3639,C 0.2919,E1 4.2282,E2 244.7655} C_DIS
LIN {X -128.776,Y -54.5869,Z 182,A -153.6904,B 4.3643,C 0.2863,E1 4.2262,E2 246.5988} C_DIS
LIN {X -129.8841,Y -51.8915,Z 182,A -155.3167,B 4.3643,C 0.2862,E1 4.2244,E2 248.2806} C_DIS
LIN {X -131.3798,Y -47.9806,Z 182,A -156.8875,B 4.3647,C 0.2807,E1 4.2229,E2 249.8319} C_DIS
LIN {X -133.0345,Y -43.1821,Z 182,A -158.8731,B 4.365,C 0.2745,E1 4.2212,E2 251.8043} C_DIS
LIN {X -134.1573,Y -39.5518,Z 182,A -160.3566,B 4.3653,C 0.2698,E1 4.22,E2 253.2774} C_DIS
LIN {X -135.099,Y -36.2044,Z 182,A -161.8865,B 4.3655,C 0.2666,E1 4.2188,E2 254.8201} C_DIS
LIN {X -136.0025,Y -32.6471,Z 182,A -163.4152,B 4.3658,C 0.2627,E1 4.2178,E2 256.3512} C_DIS
LIN {X -136.833,Y -28.9747,Z 182,A -164.987,B 4.366,C 0.2587,E1 4.2169,E2 257.9259} C_DIS
LIN {X -137.6117,Y -25.0136,Z 182,A -166.7509,B 4.3662,C 0.2548,E1 4.2159,E2 259.7031} C_DIS
LIN {X -138.1834,Y -21.6315,Z 182,A -168.1878,B 4.3665,C 0.2511,E1 4.2153,E2 261.1431} C_DIS
LIN {X -138.6271,Y -18.5804,Z 182,A -169.675,B 4.3665,C 0.2491,E1 4.2147,E2 262.6584} C_DIS
LIN {X -139.4439,Y -10.8832,Z 182,A -172.8471,B 4.3671,C 0.2402,E1 4.2139,E2 265.8286} C_DIS
LIN {X -139.8256,Y -3.4086,Z 182,A -176.9329,B 4.3671,C 0.2382,E1 4.2135,E2 270.0419} C_DIS
LIN {X -139.8185,Y 3.6642,Z 182,A -178.6742,B 4.368,C 0.2224,E1 4.2135,E2 271.6341} C_DIS
LIN {X -139.692,Y 6.9792,Z 182,A 179.3801,B 4.368,C 0.2224,E1 4.2138,E2 273.6539} C_DIS
LIN {X -139.488,Y 10.2797,Z 182,A 178.5306,B 4.3684,C 0.2153,E1 4.2139,E2 274.4378} C_DIS
LIN {X -138.883,Y 16.5542,Z 182,A 175.6126,B 4.3686,C 0.2102,E1 4.2148,E2 277.397} C_DIS
LIN {X -138.396,Y 20.2304,Z 182,A 174.1438,B 4.3688,C 0.2056,E1 4.2153,E2 278.8583} C_DIS
LIN {X -137.9501,Y 23.0712,Z 182,A 172.8459,B 4.3689,C 0.2031,E1 4.2159,E2 280.1705} C_DIS
LIN {X -136.7658,Y 29.2861,Z 182,A 170.1305,B 4.3692,C 0.1967,E1 4.2174,E2 282.8997} C_DIS
LIN {X -136.0111,Y 32.6112,Z 182,A 168.7001,B 4.3694,C 0.1931,E1 4.2183,E2 284.3333} C_DIS
LIN {X -135.2357,Y 35.692,Z 182,A 167.3049,B 4.3695,C 0.1901,E1 4.2192,E2 285.7393} C_DIS
LIN {X -134.311,Y 39.0271,Z 182,A 165.9189,B 4.3697,C 0.186,E1 4.2203,E2 287.1202} C_DIS
LIN {X -133.3031,Y 42.3414,Z 182,A 164.383,B 4.3698,C 0.183,E1 4.2216,E2 288.6697} C_DIS
LIN {X -132.2643,Y 45.4834,Z 182,A 163.1627,B 4.37,C 0.1784,E1 4.2226,E2 289.8718} C_DIS
LIN {X -131.1205,Y 48.6829,Z 182,A 161.7586,B 4.3702,C 0.1748,E1 4.224,E2 291.2763} C_DIS
LIN {X -129.639,Y 52.4998,Z 182,A 159.6766,B 4.3702,C 0.1731,E1 4.2262,E2 293.4081} C_DIS
LIN {X -127.8278,Y 56.7681,Z 182,A 157.8802,B 4.3705,C 0.1675,E1 4.2281,E2 295.19} C_DIS
LIN {X -125.8686,Y 60.9927,Z 182,A 155.5748,B 4.3705,C 0.1653,E1 4.231,E2 297.5439} C_DIS
LIN {X -124.2644,Y 64.1972,Z 182,A 154.1668,B 4.3707,C 0.1612,E1 4.2328,E2 298.9431} C_DIS
LIN {X -121.6953,Y 68.9449,Z 182,A 152.0302,B 4.3709,C 0.1552,E1 4.2356,E2 301.0686} C_DIS
LIN {X -119.495,Y 72.6916,Z 182,A 150.188,B 4.371,C 0.1514,E1 4.2383,E2 302.9171} C_DIS
LIN {X -117.139,Y 76.4299,Z 182,A 148.3299,B 4.3712,C 0.1474,E1 4.2411,E2 304.7797} C_DIS
LIN {X -114.6055,Y 80.1791,Z 182,A 146.4728,B 4.3713,C 0.1431,E1 4.244,E2 306.6357} C_DIS
LIN {X -112.5675,Y 83.0156,Z 182,A 144.6328,B 4.3713,C 0.1428,E1 4.2472,E2 308.5256} C_DIS
LIN {X -110.1144,Y 86.2429,Z 182,A 143.2552,B 4.3715,C 0.1371,E1 4.2495,E2 309.8665} C_DIS
LIN {X -107.3044,Y 89.7151,Z 182,A 141.5257,B 4.3717,C 0.1324,E1 4.2525,E2 311.582} C_DIS
LIN {X -103.9338,Y 93.599,Z 182,A 138.6851,B 4.3717,C 0.1333,E1 4.2579,E2 314.5122} C_DIS
LIN {X -100.4123,Y 97.3671,Z 182,A 137.0874,B 4.3719,C 0.1252,E1 4.2609,E2 316.0443} C_DIS
LIN {X -98.3715,Y 99.4289,Z 182,A 135.2388,B 4.3718,C 0.1278,E1 4.2648,E2 317.9739} C_DIS
LIN {X -94.3733,Y 103.2315,Z 182,A 133.0189,B 4.3719,C 0.1232,E1 4.2693,E2 320.187} C_DIS
LIN {X -90.612,Y 106.5479,Z 182,A 131.4668,B 4.3721,C 0.1157,E1 4.2724,E2 321.6753} C_DIS
LIN {X -87.2409,Y 109.3254,Z 182,A 129.6358,B 4.3721,C 0.1129,E1 4.2764,E2 323.5101} C_DIS
LIN {X -84.3443,Y 111.5752,Z 182,A 127.5996,B 4.3721,C 0.1145,E1 4.2811,E2 325.6113} C_DIS
LIN {X -80.4369,Y 114.4243,Z 182,A 126.0658,B 4.3723,C 0.1079,E1 4.2845,E2 327.0883} C_DIS
LIN {X -76.6055,Y 117.0244,Z 182,A 124.1231,B 4.3723,C 0.1053,E1 4.289,E2 329.0353} C_DIS
LIN {X -72.8104,Y 119.4227,Z 182,A 122.2791,B 4.3724,C 0.1027,E1 4.2934,E2 330.8785} C_DIS
LIN {X -68.7611,Y 121.7989,Z 182,A 120.2855,B 4.3724,C 0.1006,E1 4.2982,E2 332.8794} C_DIS
LIN {X -64.9569,Y 123.8669,Z 182,A 118.6057,B 4.3726,C 0.0976,E1 4.3023,E2 334.5462} C_DIS
LIN {X -62.0278,Y 125.3594,Z 182,A 117.2462,B 4.3726,C 0.096,E1 4.3057,E2 335.9064} C_DIS
LIN {X -58.3155,Y 127.1295,Z 182,A 115.4343,B 4.3726,C 0.0952,E1 4.3103,E2 337.7329} C_DIS
LIN {X -55.1502,Y 128.5342,Z 182,A 113.699,B 4.3726,C 0.0963,E1 4.3149,E2 339.5064} C_DIS
LIN {X -51.5114,Y 130.0367,Z 182,A 112.1741,B 4.3726,C 0.0939,E1 4.3188,E2 341.0195} C_DIS
LIN {X -48.5215,Y 131.1809,Z 182,A 110.999,B 4.3726,C 0.0916,E1 4.3218,E2 342.1769} C_DIS
LIN {X -44.539,Y 132.5853,Z 182,A 109.3583,B 4.3727,C 0.0893,E1 4.3261,E2 343.8053} C_DIS
LIN {X -41.3978,Y 133.5999,Z 182,A 107.9448,B 4.3727,C 0.0888,E1 4.3299,E2 345.2256} C_DIS
LIN {X -38.3986,Y 134.4938,Z 182,A 106.2332,B 4.3727,C 0.0916,E1 4.3347,E2 346.9895} C_DIS
LIN {X -34.2663,Y 135.6035,Z 182,A 104.955,B 4.3728,C 0.0863,E1 4.338,E2 348.2081} C_DIS
LIN {X -30.6129,Y 136.4758,Z 182,A 103.3203,B 4.3728,C 0.0863,E1 4.3424,E2 349.8538} C_DIS
LIN {X -27.0863,Y 137.2205,Z 182,A 101.8318,B 4.3728,C 0.0857,E1 4.3465,E2 351.343} C_DIS
LIN {X -19.2807,Y 138.5317,Z 182,A 98.5408,B 4.3728,C 0.0849,E1 4.3556,E2 354.6384} C_DIS
LIN {X -14.0542,Y 139.16,Z 182,A 96.215,B 4.3728,C 0.0859,E1 4.3621,E2 356.984} C_DIS
LIN {X -10.7856,Y 139.451,Z 182,A 95.1316,B 4.3728,C 0.0833,E1 4.3651,E2 358.0346} C_DIS
LIN {X -7.4246,Y 139.6696,Z 182,A 93.7029,B 4.3728,C 0.0836,E1 4.369,E2 359.4686} C_DIS
LIN {X -3.4288,Y 139.825,Z 182,A 92.0523,B 4.3728,C 0.0836,E1 4.3737,E2 361.1201} C_DIS
LIN {X 0.7279,Y 139.8644,Z 182,A 90.4077,B 4.3728,C 0.0832,E1 4.3782,E2 362.7567} C_DIS
LIN {X 4.9095,Y 139.7811,Z 182,A 88.68,B 4.3728,C 0.0836,E1 4.3831,E2 364.4855} C_DIS
LIN {X 8.7409,Y 139.5929,Z 182,A 87.1128,B 4.3728,C 0.0839,E1 4.3874,E2 366.0514} C_DIS
LIN {X 12.9239,Y 139.2685,Z 182,A 85.4295,B 4.3728,C 0.0841,E1 4.3921,E2 367.7297} C_DIS
LIN {X 16.425,Y 138.8984,Z 182,A 84.0426,B 4.3728,C 0.0841,E1 4.3959,E2 369.1092} C_DIS
LIN {X 20.5052,Y 138.3564,Z 182,A 82.0484,B 4.3728,C 0.088,E1 4.4016,E2 371.1411} C_DIS
LIN {X 23.8284,Y 137.8238,Z 182,A 80.8348,B 4.3728,C 0.0871,E1 4.4048,E2 372.3339} C_DIS
LIN {X 27.2306,Y 137.1913,Z 182,A 79.548,B 4.3728,C 0.0866,E1 4.4083,E2 373.6041} C_DIS
LIN {X 30.8309,Y 136.426,Z 182,A 77.9487,B 4.3728,C 0.0885,E1 4.4127,E2 375.2143} C_DIS
LIN {X 35.5471,Y 135.2743,Z 182,A 76.1107,B 4.3728,C 0.0885,E1 4.4177,E2 377.033} C_DIS
LIN {X 38.617,Y 134.431,Z 182,A 74.7366,B 4.3728,C 0.0903,E1 4.4214,E2 378.4156} C_DIS
LIN {X 41.2152,Y 133.6557,Z 182,A 73.0317,B 4.3726,C 0.0975,E1 4.4261,E2 380.1936} C_DIS
LIN {X 46.4089,Y 131.9434,Z 182,A 71.3548,B 4.3726,C 0.0938,E1 4.4304,E2 381.8006} C_DIS
LIN {X 50.0389,Y 130.6101,Z 182,A 69.8287,B 4.3726,C 0.0948,E1 4.4343,E2 383.3193} C_DIS
LIN {X 53.5763,Y 129.1981,Z 182,A 68.339,B 4.3726,C 0.0958,E1 4.4382,E2 384.7999} C_DIS
LIN {X 56.9931,Y 127.7271,Z 182,A 66.9693,B 4.3726,C 0.096,E1 4.4416,E2 386.1502} C_DIS
LIN {X 62.6719,Y 125.0416,Z 182,A 64.3318,B 4.3726,C 0.1,E1 4.4483,E2 388.7956} C_DIS
LIN {X 66.07,Y 123.2792,Z 182,A 62.7114,B 4.3724,C 0.1027,E1 4.4523,E2 390.4224} C_DIS
LIN {X 69.9467,Y 121.1217,Z 182,A 60.9102,B 4.3724,C 0.1051,E1 4.4567,E2 392.2215} C_DIS
LIN {X 73.9401,Y 118.7259,Z 182,A 59.055,B 4.3724,C 0.1075,E1 4.4611,E2 394.0701} C_DIS
LIN {X 77.7893,Y 116.2404,Z 182,A 56.9567,B 4.3722,C 0.113,E1 4.466,E2 396.1961} C_DIS
LIN {X 80.7355,Y 114.2137,Z 182,A 55.7226,B 4.3722,C 0.1128,E1 4.4688,E2 397.4014} C_DIS
LIN {X 84.6035,Y 111.3796,Z 182,A 53.7948,B 4.3722,C 0.1158,E1 4.4731,E2 399.3248} C_DIS
LIN {X 88.1902,Y 108.5617,Z 182,A 51.9359,B 4.372,C 0.119,E1 4.4772,E2 401.1827} C_DIS
LIN {X 91.904,Y 105.4355,Z 182,A 50.1014,B 4.372,C 0.121,E1 4.481,E2 402.9981} C_DIS
LIN {X 94.5896,Y 103.033,Z 182,A 48.0645,B 4.3717,C 0.1304,E1 4.4854,E2 405.1054} C_DIS
LIN {X 98.4524,Y 99.3486,Z 182,A 46.4866,B 4.3717,C 0.1276,E1 4.4883,E2 406.6075} C_DIS
LIN {X 101.5527,Y 96.1774,Z 182,A 44.854,B 4.3717,C 0.1292,E1 4.4915,E2 408.2173} C_DIS
LIN {X 104.0552,Y 93.464,Z 182,A 43.2215,B 4.3717,C 0.1338,E1 4.4946,E2 409.8653} C_DIS
LIN {X 107.1441,Y 89.9061,Z 182,A 41.0073,B 4.3714,C 0.1415,E1 4.4986,E2 412.1157} C_DIS
LIN {X 109.7787,Y 86.6703,Z 182,A 39.642,B 4.3714,C 0.1411,E1 4.5009,E2 413.4382} C_DIS
LIN {X 112.6007,Y 82.9705,Z 182,A 37.8108,B 4.3713,C 0.1446,E1 4.504,E2 415.2605} C_DIS
LIN {X 115.2365,Y 79.2689,Z 182,A 36.0132,B 4.3711,C 0.1482,E1 4.5069,E2 417.0505} C_DIS
LIN {X 117.7317,Y 75.5133,Z 182,A 34.2089,B 4.3711,C 0.152,E1 4.5096,E2 418.85} C_DIS
LIN {X 121.0994,Y 69.985,Z 182,A 31.5673,B 4.3708,C 0.1584,E1 4.5134,E2 421.4913} C_DIS
LIN {X 123.3773,Y 65.8875,Z 182,A 29.7222,B 4.3706,C 0.1622,E1 4.5158,E2 423.3278} C_DIS
LIN {X 125.2804,Y 62.1882,Z 182,A 28.2258,B 4.3706,C 0.164,E1 4.5177,E2 424.7983} C_DIS
LIN {X 126.8002,Y 59.0275,Z 182,A 26.8045,B 4.3705,C 0.1675,E1 4.5194,E2 426.2183} C_DIS
LIN {X 128.1551,Y 56.027,Z 182,A 25.6001,B 4.3704,C 0.1691,E1 4.5207,E2 427.4049} C_DIS
LIN {X 130.2131,Y 51.0593,Z 182,A 23.1632,B 4.37,C 0.1779,E1 4.5234,E2 429.8727} C_DIS
LIN {X 132.0261,Y 46.1703,Z 182,A 21.2876,B 4.37,C 0.1803,E1 4.5251,E2 431.7162} C_DIS
LIN {X 133.1203,Y 42.9137,Z 182,A 19.924,B 4.3698,C 0.1835,E1 4.5263,E2 433.0749} C_DIS
LIN {X 134.1132,Y 39.7026,Z 182,A 18.6207,B 4.3697,C 0.1863,E1 4.5273,E2 434.3696} C_DIS
LIN {X 135.1264,Y 36.1019,Z 182,A 17.1827,B 4.3696,C 0.1893,E1 4.5284,E2 435.7962} C_DIS
LIN {X 135.8688,Y 33.2014,Z 182,A 15.7968,B 4.3693,C 0.1947,E1 4.5293,E2 437.2034} C_DIS
LIN {X 136.7228,Y 29.485,Z 182,A 14.0131,B 4.369,C 0.2019,E1 4.5304,E2 439.0164} C_DIS
LIN {X 137.5282,Y 25.4783,Z 182,A 12.6894,B 4.369,C 0.202,E1 4.5311,E2 440.2963} C_DIS
LIN {X 138.7621,Y 17.5461,Z 182,A 9.5097,B 4.3686,C 0.2099,E1 4.5324,E2 443.4641} C_DIS
LIN {X 139.2169,Y 13.4619,Z 182,A 7.9295,B 4.3685,C 0.2133,E1 4.5328,E2 445.0321} C_DIS
Enddeposition()
END
